SPLINE
SPL {X   -94.059, Y  +248.080, Z    +0.000, E1   +58.275, E3 +53997.383}
SPL {X  -130.769, Y  +285.325, Z    +0.000, E1   +56.495, E3 +54037.260}
SPL {X  -149.689, Y  +321.019, Z    +0.000, E1   +46.817, E3 +54049.344}
SPL {X  -157.484, Y  +349.293, Z    +0.000, E1   +30.654, E3 +54053.637}
SPL {X  -159.556, Y  +365.719, Z    +0.000, E1   +15.845, E3 +54054.829}
SPL {X  -159.982, Y  +375.924, Z    +0.000, E1    +4.476, E3 +54055.131}
SPL {X  -159.990, Y  +379.531, Z    +0.000, E1    -0.039, E3 +54055.158}
SPL {X  -159.990, Y  +382.420, Z    +0.000, E1    -7.600, E3 +54055.186}
SPL {X  -159.990, Y  +386.504, Z    +0.000, E1   -19.860, E3 +54055.292}
SPL {X  -159.990, Y  +392.530, Z    +0.000, E1   -36.133, E3 +54055.607}
SPL {X  -159.990, Y  +400.492, Z    +0.000, E1   -51.837, E3 +54056.260}
SPL {X  -159.990, Y  +409.662, Z    +0.000, E1   -61.705, E3 +54057.371}
SPL {X  -159.990, Y  +434.697, Z    +0.000, E1   -71.504, E3 +54062.391}
SPL {X  -159.990, Y  +521.523, Z    +0.000, E1   -76.035, E3 +54088.671}
SPL {X  -154.459, Y  +718.205, Z    +0.000, E1   -76.329, E3 +54170.467}
SPL {X  -151.356, Y  +728.349, Z    +0.000, E1   -76.056, E3 +54178.682}
SPL {X  -147.124, Y  +739.360, Z    +0.000, E1   -75.690, E3 +54188.278}
SPL {X  -142.861, Y  +748.524, Z    +0.000, E1   -75.261, E3 +54196.963}
SPL {X  -138.117, Y  +757.250, Z    +0.000, E1   -74.803, E3 +54205.567}
SPL {X  -133.491, Y  +764.686, Z    +0.000, E1   -74.276, E3 +54213.308}
SPL {X  -128.839, Y  +771.354, Z    +0.000, E1   -73.759, E3 +54220.326}
SPL {X  -124.765, Y  +776.652, Z    +0.000, E1   -73.233, E3 +54225.976}
SPL {X  -121.376, Y  +780.734, Z    +0.000, E1   -72.804, E3 +54230.238}
SPL {X  -118.281, Y  +784.233, Z    +0.000, E1   -72.371, E3 +54233.806}
SPL {X   -72.391, Y  +819.176, Z    +0.000, E1   -59.867, E3 +54329.692}
ENDSPLINE

SPLINE
SPL {X  -116.241, Y  +786.431, Z    +0.000, E1   -57.120, E3 +54554.134}
SPL {X  -148.710, Y  +735.509, Z    +0.000, E1   -46.282, E3 +54579.867}
SPL {X  -157.559, Y  +704.285, Z    +0.000, E1   -29.037, E3 +54585.196}
SPL {X  -159.709, Y  +685.986, Z    +0.000, E1   -12.810, E3 +54586.528}
SPL {X  -159.990, Y  +674.648, Z    +0.000, E1    -0.349, E3 +54586.787}
SPL {X  -159.990, Y  +672.787, Z    +0.000, E1    +4.022, E3 +54586.800}
SPL {X  -159.990, Y  +669.267, Z    +0.000, E1   +13.665, E3 +54586.870}
SPL {X  -159.990, Y  +663.438, Z    +0.000, E1   +29.379, E3 +54587.141}
SPL {X  -159.990, Y  +655.264, Z    +0.000, E1   +47.291, E3 +54587.758}
SPL {X  -159.990, Y  +645.368, Z    +0.000, E1   +59.257, E3 +54589.001}
SPL {X  -159.990, Y  +624.023, Z    +0.000, E1   +69.513, E3 +54593.126}
SPL {X  -159.990, Y  +543.075, Z    +0.000, E1   +75.590, E3 +54616.774}
SPL {X  -156.121, Y  +342.530, Z    +0.000, E1   +75.868, E3 +54703.420}
SPL {X  -153.498, Y  +332.386, Z    +0.000, E1   +75.628, E3 +54711.425}
ENDSPLINE

SPLINE
SPL {X  -155.252, Y  +338.851, Z    +0.000, E1   +74.632, E3 +54718.803}
SPL {X  -159.103, Y  +360.678, Z    +0.000, E1   +72.233, E3 +54731.128}
ENDSPLINE

SPLINE
SPL {X  -154.371, Y  +335.471, Z    +0.000, E1   +73.016, E3 +54739.698}
SPL {X  -149.938, Y  +321.685, Z    +0.000, E1   +73.398, E3 +54744.393}
SPL {X  -145.016, Y  +309.920, Z    +0.000, E1   +73.647, E3 +54748.914}
SPL {X  -136.944, Y  +294.777, Z    +0.000, E1   +74.219, E3 +54752.215}
SPL {X  -132.590, Y  +287.964, Z    +0.000, E1   +73.910, E3 +54757.960}
SPL {X  -129.541, Y  +283.606, Z    +0.000, E1   +73.551, E3 +54762.600}
SPL {X  -125.403, Y  +278.147, Z    +0.000, E1   +73.063, E3 +54768.407}
SPL {X  -121.908, Y  +273.889, Z    +0.000, E1   +72.578, E3 +54772.954}
SPL {X  -119.156, Y  +270.736, Z    +0.000, E1   +72.213, E3 +54776.204}
SPL {X  -117.531, Y  +268.949, Z    +0.000, E1   +71.964, E3 +54778.019}
SPL {X   -74.907, Y  +236.129, Z    +0.000, E1   +61.720, E3 +54855.055}
ENDSPLINE

SPLINE
SPL {X   -94.059, Y  +248.080, Z    +0.000, E1   +58.275, E3 +55076.748}
SPL {X  -130.769, Y  +285.325, Z    +0.000, E1   +56.495, E3 +55116.625}
SPL {X  -149.689, Y  +321.019, Z    +0.000, E1   +46.817, E3 +55128.709}
SPL {X  -155.950, Y  +341.772, Z    +0.000, E1   +35.915, E3 +55132.208}
SPL {X  -158.168, Y  +353.421, Z    +0.000, E1   +27.296, E3 +55133.393}
SPL {X  -159.556, Y  +365.719, Z    +0.000, E1   +15.845, E3 +55134.194}
SPL {X  -159.982, Y  +375.924, Z    +0.000, E1    +4.476, E3 +55134.496}
SPL {X  -159.990, Y  +379.800, Z    +0.000, E1    -0.377, E3 +55134.524}
SPL {X  -159.990, Y  +383.422, Z    +0.000, E1   -10.730, E3 +55134.567}
SPL {X  -159.990, Y  +387.978, Z    +0.000, E1   -23.882, E3 +55134.720}
SPL {X  -159.990, Y  +394.494, Z    +0.000, E1   -40.961, E3 +55135.101}
SPL {X  -159.990, Y  +400.492, Z    +0.000, E1   -51.837, E3 +55135.625}
SPL {X  -159.990, Y  +409.662, Z    +0.000, E1   -61.705, E3 +55136.736}
SPL {X  -159.990, Y  +434.697, Z    +0.000, E1   -71.504, E3 +55141.756}
SPL {X  -159.990, Y  +521.523, Z    +0.000, E1   -76.035, E3 +55168.036}
SPL {X  -154.459, Y  +718.205, Z    +0.000, E1   -76.329, E3 +55249.832}
SPL {X  -151.356, Y  +728.349, Z    +0.000, E1   -76.056, E3 +55258.047}
SPL {X  -147.124, Y  +739.360, Z    +0.000, E1   -75.690, E3 +55267.644}
SPL {X  -142.861, Y  +748.524, Z    +0.000, E1   -75.261, E3 +55276.328}
SPL {X  -138.117, Y  +757.250, Z    +0.000, E1   -74.803, E3 +55284.932}
SPL {X  -133.491, Y  +764.686, Z    +0.000, E1   -74.276, E3 +55292.673}
SPL {X  -130.530, Y  +769.013, Z    +0.000, E1   -73.929, E3 +55297.255}
SPL {X  -127.734, Y  +772.837, Z    +0.000, E1   -73.601, E3 +55301.307}
SPL {X  -124.765, Y  +776.652, Z    +0.000, E1   -73.233, E3 +55305.341}
SPL {X  -121.376, Y  +780.734, Z    +0.000, E1   -72.804, E3 +55309.603}
SPL {X  -118.281, Y  +784.233, Z    +0.000, E1   -72.371, E3 +55313.171}
SPL {X   -72.391, Y  +819.176, Z    +0.000, E1   -59.867, E3 +55409.057}
ENDSPLINE

SPLINE
SPL {X  -116.241, Y  +786.431, Z    +0.000, E1   -57.120, E3 +55633.499}
SPL {X  -148.710, Y  +735.509, Z    +0.000, E1   -46.282, E3 +55659.232}
SPL {X  -157.559, Y  +704.285, Z    +0.000, E1   -29.037, E3 +55664.561}
SPL {X  -159.430, Y  +689.871, Z    +0.000, E1   -16.582, E3 +55665.711}
SPL {X  -159.960, Y  +679.609, Z    +0.000, E1    -6.021, E3 +55666.094}
SPL {X  -159.990, Y  +674.508, Z    +0.000, E1    -0.018, E3 +55666.153}
SPL {X  -159.990, Y  +672.787, Z    +0.000, E1    +4.022, E3 +55666.165}
SPL {X  -159.990, Y  +669.267, Z    +0.000, E1   +13.665, E3 +55666.235}
SPL {X  -159.990, Y  +663.438, Z    +0.000, E1   +29.379, E3 +55666.506}
SPL {X  -159.990, Y  +655.264, Z    +0.000, E1   +47.291, E3 +55667.123}
SPL {X  -159.990, Y  +645.368, Z    +0.000, E1   +59.257, E3 +55668.366}
SPL {X  -159.990, Y  +624.023, Z    +0.000, E1   +69.513, E3 +55672.491}
SPL {X  -159.990, Y  +543.075, Z    +0.000, E1   +75.590, E3 +55696.139}
SPL {X  -156.121, Y  +342.530, Z    +0.000, E1   +75.868, E3 +55782.785}
SPL {X  -153.498, Y  +332.386, Z    +0.000, E1   +75.628, E3 +55790.790}
ENDSPLINE

SPLINE
SPL {X  -155.252, Y  +338.851, Z    +0.000, E1   +74.632, E3 +55798.168}
SPL {X  -159.103, Y  +360.678, Z    +0.000, E1   +72.233, E3 +55810.493}
ENDSPLINE

SPLINE
SPL {X  -154.371, Y  +335.471, Z    +0.000, E1   +73.016, E3 +55819.064}
SPL {X  -149.938, Y  +321.685, Z    +0.000, E1   +73.398, E3 +55823.758}
SPL {X  -145.016, Y  +309.920, Z    +0.000, E1   +73.647, E3 +55828.279}
SPL {X  -139.138, Y  +298.522, Z    +0.000, E1   +74.138, E3 +55830.295}
SPL {X  -135.697, Y  +292.747, Z    +0.000, E1   +74.259, E3 +55832.297}
SPL {X  -132.590, Y  +287.964, Z    +0.000, E1   +73.910, E3 +55837.325}
SPL {X  -129.541, Y  +283.606, Z    +0.000, E1   +73.551, E3 +55841.965}
SPL {X  -126.457, Y  +279.493, Z    +0.000, E1   +73.175, E3 +55846.364}
SPL {X  -122.770, Y  +274.912, Z    +0.000, E1   +72.712, E3 +55851.220}
SPL {X  -119.156, Y  +270.736, Z    +0.000, E1   +72.213, E3 +55855.569}
SPL {X  -117.531, Y  +268.949, Z    +0.000, E1   +71.964, E3 +55857.384}
SPL {X   -74.907, Y  +236.129, Z    +0.000, E1   +61.720, E3 +55934.420}
ENDSPLINE

SPLINE
SPL {X   -94.059, Y  +248.080, Z    +0.000, E1   +58.275, E3 +56156.113}
SPL {X  -130.769, Y  +285.325, Z    +0.000, E1   +56.495, E3 +56195.990}
SPL {X  -149.689, Y  +321.019, Z    +0.000, E1   +46.817, E3 +56208.074}
SPL {X  -157.484, Y  +349.293, Z    +0.000, E1   +30.654, E3 +56212.367}
SPL {X  -159.556, Y  +365.719, Z    +0.000, E1   +15.845, E3 +56213.559}
SPL {X  -159.982, Y  +375.924, Z    +0.000, E1    +4.476, E3 +56213.861}
SPL {X  -159.990, Y  +379.531, Z    +0.000, E1    -0.039, E3 +56213.888}
SPL {X  -159.990, Y  +382.420, Z    +0.000, E1    -7.600, E3 +56213.916}
SPL {X  -159.990, Y  +386.504, Z    +0.000, E1   -19.860, E3 +56214.022}
SPL {X  -159.990, Y  +392.530, Z    +0.000, E1   -36.133, E3 +56214.337}
SPL {X  -159.990, Y  +400.492, Z    +0.000, E1   -51.837, E3 +56214.990}
SPL {X  -159.990, Y  +409.662, Z    +0.000, E1   -61.705, E3 +56216.101}
SPL {X  -159.990, Y  +434.697, Z    +0.000, E1   -71.504, E3 +56221.121}
SPL {X  -159.990, Y  +521.523, Z    +0.000, E1   -76.035, E3 +56247.401}
SPL {X  -154.459, Y  +718.205, Z    +0.000, E1   -76.329, E3 +56329.197}
SPL {X  -151.356, Y  +728.349, Z    +0.000, E1   -76.056, E3 +56337.412}
SPL {X  -148.399, Y  +736.287, Z    +0.000, E1   -75.788, E3 +56344.291}
SPL {X  -144.005, Y  +746.209, Z    +0.000, E1   -75.396, E3 +56353.407}
SPL {X  -138.117, Y  +757.250, Z    +0.000, E1   -74.803, E3 +56364.297}
SPL {X  -133.491, Y  +764.686, Z    +0.000, E1   -74.276, E3 +56372.038}
SPL {X  -128.839, Y  +771.354, Z    +0.000, E1   -73.759, E3 +56379.057}
SPL {X  -123.568, Y  +778.125, Z    +0.000, E1   -73.105, E3 +56386.228}
SPL {X  -118.985, Y  +783.455, Z    +0.000, E1   -72.490, E3 +56391.736}
SPL {X   -72.391, Y  +819.176, Z    +0.000, E1   -59.867, E3 +56488.422}
ENDSPLINE

SPLINE
SPL {X   -92.809, Y  +806.820, Z    +0.000, E1   -56.994, E3 +56681.217}
SPL {X  -120.521, Y  +781.721, Z    +0.000, E1   -56.766, E3 +56717.316}
SPL {X  -143.482, Y  +747.279, Z    +0.000, E1   -50.227, E3 +56735.329}
SPL {X  -154.118, Y  +719.449, Z    +0.000, E1   -38.836, E3 +56741.908}
SPL {X  -158.958, Y  +694.646, Z    +0.000, E1   -21.132, E3 +56744.760}
SPL {X  -159.960, Y  +679.609, Z    +0.000, E1    -6.021, E3 +56745.460}
SPL {X  -159.990, Y  +674.508, Z    +0.000, E1    -0.018, E3 +56745.518}
SPL {X  -159.990, Y  +672.787, Z    +0.000, E1    +4.022, E3 +56745.530}
SPL {X  -159.990, Y  +669.267, Z    +0.000, E1   +13.665, E3 +56745.600}
SPL {X  -159.990, Y  +663.438, Z    +0.000, E1   +29.379, E3 +56745.871}
SPL {X  -159.990, Y  +655.264, Z    +0.000, E1   +47.291, E3 +56746.488}
SPL {X  -159.990, Y  +645.368, Z    +0.000, E1   +59.257, E3 +56747.731}
SPL {X  -159.990, Y  +624.023, Z    +0.000, E1   +69.513, E3 +56751.856}
SPL {X  -159.990, Y  +543.075, Z    +0.000, E1   +75.590, E3 +56775.504}
SPL {X  -156.121, Y  +342.530, Z    +0.000, E1   +75.868, E3 +56862.150}
SPL {X  -153.498, Y  +332.386, Z    +0.000, E1   +75.628, E3 +56870.155}
ENDSPLINE

SPLINE
SPL {X  -155.252, Y  +338.851, Z    +0.000, E1   +74.632, E3 +56877.533}
SPL {X  -159.103, Y  +360.678, Z    +0.000, E1   +72.233, E3 +56889.858}
ENDSPLINE

SPLINE
SPL {X  -154.371, Y  +335.471, Z    +0.000, E1   +73.016, E3 +56898.429}
SPL {X  -149.938, Y  +321.685, Z    +0.000, E1   +73.398, E3 +56903.123}
SPL {X  -145.016, Y  +309.920, Z    +0.000, E1   +73.647, E3 +56907.644}
SPL {X  -139.138, Y  +298.522, Z    +0.000, E1   +74.138, E3 +56909.660}
SPL {X  -135.697, Y  +292.747, Z    +0.000, E1   +74.259, E3 +56911.662}
SPL {X  -132.590, Y  +287.964, Z    +0.000, E1   +73.910, E3 +56916.690}
SPL {X  -129.541, Y  +283.606, Z    +0.000, E1   +73.551, E3 +56921.330}
SPL {X  -126.457, Y  +279.493, Z    +0.000, E1   +73.175, E3 +56925.729}
SPL {X  -122.770, Y  +274.912, Z    +0.000, E1   +72.712, E3 +56930.585}
SPL {X  -118.941, Y  +270.496, Z    +0.000, E1   +72.188, E3 +56935.172}
SPL {X   -74.907, Y  +236.129, Z    +0.000, E1   +61.720, E3 +57013.785}
ENDSPLINE

SPLINE
SPL {X   -94.059, Y  +248.080, Z    +0.000, E1   +58.275, E3 +57235.478}
SPL {X  -136.558, Y  +294.141, Z    +0.000, E1   +54.887, E3 +57279.333}
SPL {X  -151.843, Y  +327.098, Z    +0.000, E1   +44.118, E3 +57288.692}
SPL {X  -157.484, Y  +349.293, Z    +0.000, E1   +30.654, E3 +57291.732}
SPL {X  -159.556, Y  +365.719, Z    +0.000, E1   +15.845, E3 +57292.924}
SPL {X  -159.982, Y  +375.924, Z    +0.000, E1    +4.476, E3 +57293.226}
SPL {X  -159.990, Y  +379.531, Z    +0.000, E1    -0.039, E3 +57293.253}
SPL {X  -159.990, Y  +382.420, Z    +0.000, E1    -7.600, E3 +57293.281}
SPL {X  -159.990, Y  +386.504, Z    +0.000, E1   -19.860, E3 +57293.387}
SPL {X  -159.990, Y  +392.530, Z    +0.000, E1   -36.133, E3 +57293.702}
SPL {X  -159.990, Y  +400.492, Z    +0.000, E1   -51.837, E3 +57294.355}
SPL {X  -159.990, Y  +409.662, Z    +0.000, E1   -61.705, E3 +57295.466}
SPL {X  -159.990, Y  +434.697, Z    +0.000, E1   -71.504, E3 +57300.486}
SPL {X  -159.990, Y  +521.523, Z    +0.000, E1   -76.035, E3 +57326.767}
SPL {X  -154.459, Y  +718.205, Z    +0.000, E1   -76.329, E3 +57408.562}
SPL {X  -151.356, Y  +728.349, Z    +0.000, E1   -76.056, E3 +57416.777}
SPL {X  -148.399, Y  +736.287, Z    +0.000, E1   -75.788, E3 +57423.656}
SPL {X  -144.005, Y  +746.209, Z    +0.000, E1   -75.396, E3 +57432.772}
SPL {X  -138.117, Y  +757.250, Z    +0.000, E1   -74.803, E3 +57443.662}
SPL {X  -133.491, Y  +764.686, Z    +0.000, E1   -74.276, E3 +57451.403}
SPL {X  -128.839, Y  +771.354, Z    +0.000, E1   -73.759, E3 +57458.422}
SPL {X  -123.568, Y  +778.125, Z    +0.000, E1   -73.105, E3 +57465.593}
SPL {X  -118.985, Y  +783.455, Z    +0.000, E1   -72.490, E3 +57471.101}
SPL {X   -72.391, Y  +819.176, Z    +0.000, E1   -59.867, E3 +57567.787}
ENDSPLINE

SPLINE
SPL {X   -92.809, Y  +806.820, Z    +0.000, E1   -56.994, E3 +57760.582}
SPL {X  -120.521, Y  +781.721, Z    +0.000, E1   -56.766, E3 +57796.681}
SPL {X  -148.710, Y  +735.509, Z    +0.000, E1   -46.282, E3 +57817.962}
SPL {X  -157.559, Y  +704.285, Z    +0.000, E1   -29.037, E3 +57823.291}
SPL {X  -159.430, Y  +689.871, Z    +0.000, E1   -16.582, E3 +57824.442}
SPL {X  -159.960, Y  +679.609, Z    +0.000, E1    -6.021, E3 +57824.825}
SPL {X  -159.990, Y  +674.508, Z    +0.000, E1    -0.018, E3 +57824.883}
SPL {X  -159.990, Y  +672.787, Z    +0.000, E1    +4.022, E3 +57824.895}
SPL {X  -159.990, Y  +669.267, Z    +0.000, E1   +13.665, E3 +57824.965}
SPL {X  -159.990, Y  +663.438, Z    +0.000, E1   +29.379, E3 +57825.236}
SPL {X  -159.990, Y  +655.264, Z    +0.000, E1   +47.291, E3 +57825.853}
SPL {X  -159.990, Y  +645.368, Z    +0.000, E1   +59.257, E3 +57827.096}
SPL {X  -159.990, Y  +624.023, Z    +0.000, E1   +69.513, E3 +57831.221}
SPL {X  -159.990, Y  +543.075, Z    +0.000, E1   +75.590, E3 +57854.869}
SPL {X  -156.121, Y  +342.530, Z    +0.000, E1   +75.868, E3 +57941.515}
SPL {X  -153.865, Y  +333.657, Z    +0.000, E1   +75.438, E3 +57951.119}
ENDSPLINE

SPLINE
SPL {X  -159.644, Y  +366.989, Z    +0.000, E1   +72.058, E3 +57966.646}
ENDSPLINE

SPLINE
SPL {X  -156.933, Y  +346.374, Z    +0.000, E1   +72.645, E3 +57974.535}
SPL {X  -151.144, Y  +325.039, Z    +0.000, E1   +73.323, E3 +57981.215}
SPL {X  -145.016, Y  +309.920, Z    +0.000, E1   +73.647, E3 +57987.009}
SPL {X  -136.944, Y  +294.777, Z    +0.000, E1   +74.219, E3 +57990.311}
SPL {X  -132.590, Y  +287.964, Z    +0.000, E1   +73.910, E3 +57996.055}
SPL {X  -129.541, Y  +283.606, Z    +0.000, E1   +73.551, E3 +58000.695}
SPL {X  -125.403, Y  +278.147, Z    +0.000, E1   +73.063, E3 +58006.503}
SPL {X  -121.908, Y  +273.889, Z    +0.000, E1   +72.578, E3 +58011.049}
SPL {X  -118.941, Y  +270.496, Z    +0.000, E1   +72.188, E3 +58014.537}
SPL {X   -74.907, Y  +236.129, Z    +0.000, E1   +61.720, E3 +58093.150}
ENDSPLINE

SPLINE
SPL {X   -94.059, Y  +248.080, Z    +0.000, E1   +58.275, E3 +58314.843}
SPL {X  -136.558, Y  +294.141, Z    +0.000, E1   +54.887, E3 +58358.698}
SPL {X  -151.843, Y  +327.098, Z    +0.000, E1   +44.118, E3 +58368.058}
SPL {X  -157.484, Y  +349.293, Z    +0.000, E1   +30.654, E3 +58371.097}
SPL {X  -159.556, Y  +365.719, Z    +0.000, E1   +15.845, E3 +58372.289}
SPL {X  -159.982, Y  +375.924, Z    +0.000, E1    +4.476, E3 +58372.591}
SPL {X  -159.990, Y  +379.531, Z    +0.000, E1    -0.039, E3 +58372.618}
SPL {X  -159.990, Y  +382.420, Z    +0.000, E1    -7.600, E3 +58372.647}
SPL {X  -159.990, Y  +386.504, Z    +0.000, E1   -19.860, E3 +58372.752}
SPL {X  -159.990, Y  +392.530, Z    +0.000, E1   -36.133, E3 +58373.067}
SPL {X  -159.990, Y  +400.492, Z    +0.000, E1   -51.837, E3 +58373.720}
SPL {X  -159.990, Y  +409.662, Z    +0.000, E1   -61.705, E3 +58374.831}
SPL {X  -159.990, Y  +434.697, Z    +0.000, E1   -71.504, E3 +58379.851}
SPL {X  -159.990, Y  +521.523, Z    +0.000, E1   -76.035, E3 +58406.132}
SPL {X  -154.459, Y  +718.205, Z    +0.000, E1   -76.329, E3 +58487.927}
SPL {X  -151.356, Y  +728.349, Z    +0.000, E1   -76.056, E3 +58496.143}
SPL {X  -148.399, Y  +736.287, Z    +0.000, E1   -75.788, E3 +58503.021}
SPL {X  -144.005, Y  +746.209, Z    +0.000, E1   -75.396, E3 +58512.137}
SPL {X  -138.117, Y  +757.250, Z    +0.000, E1   -74.803, E3 +58523.027}
SPL {X  -133.491, Y  +764.686, Z    +0.000, E1   -74.276, E3 +58530.768}
SPL {X  -128.839, Y  +771.354, Z    +0.000, E1   -73.759, E3 +58537.787}
SPL {X  -123.568, Y  +778.125, Z    +0.000, E1   -73.105, E3 +58544.958}
SPL {X  -118.985, Y  +783.455, Z    +0.000, E1   -72.490, E3 +58550.466}
SPL {X   -72.391, Y  +819.176, Z    +0.000, E1   -59.867, E3 +58647.152}
ENDSPLINE

SPLINE
SPL {X   -92.809, Y  +806.820, Z    +0.000, E1   -56.994, E3 +58839.947}
SPL {X  -120.521, Y  +781.721, Z    +0.000, E1   -56.766, E3 +58876.046}
SPL {X  -143.482, Y  +747.279, Z    +0.000, E1   -50.227, E3 +58894.059}
SPL {X  -154.118, Y  +719.449, Z    +0.000, E1   -38.836, E3 +58900.638}
SPL {X  -158.958, Y  +694.646, Z    +0.000, E1   -21.132, E3 +58903.490}
SPL {X  -159.960, Y  +679.609, Z    +0.000, E1    -6.021, E3 +58904.190}
SPL {X  -159.990, Y  +674.508, Z    +0.000, E1    -0.018, E3 +58904.248}
SPL {X  -159.990, Y  +672.787, Z    +0.000, E1    +4.022, E3 +58904.260}
SPL {X  -159.990, Y  +669.267, Z    +0.000, E1   +13.665, E3 +58904.330}
SPL {X  -159.990, Y  +663.438, Z    +0.000, E1   +29.379, E3 +58904.601}
SPL {X  -159.990, Y  +655.264, Z    +0.000, E1   +47.291, E3 +58905.218}
SPL {X  -159.990, Y  +645.368, Z    +0.000, E1   +59.257, E3 +58906.461}
SPL {X  -159.990, Y  +624.023, Z    +0.000, E1   +69.513, E3 +58910.586}
SPL {X  -159.990, Y  +543.075, Z    +0.000, E1   +75.590, E3 +58934.234}
SPL {X  -156.121, Y  +342.530, Z    +0.000, E1   +75.868, E3 +59020.880}
SPL {X  -153.498, Y  +332.386, Z    +0.000, E1   +75.628, E3 +59028.885}
ENDSPLINE

SPLINE
SPL {X  -155.252, Y  +338.851, Z    +0.000, E1   +74.632, E3 +59036.263}
SPL {X  -159.103, Y  +360.678, Z    +0.000, E1   +72.233, E3 +59048.588}
ENDSPLINE

SPLINE
SPL {X  -154.371, Y  +335.471, Z    +0.000, E1   +73.016, E3 +59057.159}
SPL {X  -149.938, Y  +321.685, Z    +0.000, E1   +73.398, E3 +59061.853}
SPL {X  -145.016, Y  +309.920, Z    +0.000, E1   +73.647, E3 +59066.374}
SPL {X  -139.138, Y  +298.522, Z    +0.000, E1   +74.138, E3 +59068.390}
SPL {X  -135.697, Y  +292.747, Z    +0.000, E1   +74.259, E3 +59070.392}
SPL {X  -132.590, Y  +287.964, Z    +0.000, E1   +73.910, E3 +59075.420}
SPL {X  -129.541, Y  +283.606, Z    +0.000, E1   +73.551, E3 +59080.061}
SPL {X  -126.457, Y  +279.493, Z    +0.000, E1   +73.175, E3 +59084.460}
SPL {X  -122.770, Y  +274.912, Z    +0.000, E1   +72.712, E3 +59089.315}
SPL {X  -118.941, Y  +270.496, Z    +0.000, E1   +72.188, E3 +59093.902}
SPL {X   -74.907, Y  +236.129, Z    +0.000, E1   +61.720, E3 +59172.516}
ENDSPLINE

SPLINE
SPL {X   -94.059, Y  +248.080, Z    +0.000, E1   +58.275, E3 +59394.209}
SPL {X  -136.558, Y  +294.141, Z    +0.000, E1   +54.887, E3 +59438.063}
SPL {X  -151.843, Y  +327.098, Z    +0.000, E1   +44.118, E3 +59447.423}
SPL {X  -157.484, Y  +349.293, Z    +0.000, E1   +30.654, E3 +59450.462}
SPL {X  -159.556, Y  +365.719, Z    +0.000, E1   +15.845, E3 +59451.655}
SPL {X  -159.982, Y  +375.924, Z    +0.000, E1    +4.476, E3 +59451.956}
SPL {X  -159.990, Y  +379.531, Z    +0.000, E1    -0.039, E3 +59451.983}
SPL {X  -159.990, Y  +382.420, Z    +0.000, E1    -7.600, E3 +59452.012}
SPL {X  -159.990, Y  +386.504, Z    +0.000, E1   -19.860, E3 +59452.117}
SPL {X  -159.990, Y  +392.530, Z    +0.000, E1   -36.133, E3 +59452.432}
SPL {X  -159.990, Y  +400.492, Z    +0.000, E1   -51.837, E3 +59453.085}
SPL {X  -159.990, Y  +409.662, Z    +0.000, E1   -61.705, E3 +59454.196}
SPL {X  -159.990, Y  +434.697, Z    +0.000, E1   -71.504, E3 +59459.216}
SPL {X  -159.990, Y  +521.523, Z    +0.000, E1   -76.035, E3 +59485.497}
SPL {X  -154.459, Y  +718.205, Z    +0.000, E1   -76.329, E3 +59567.292}
SPL {X  -151.356, Y  +728.349, Z    +0.000, E1   -76.056, E3 +59575.508}
SPL {X  -148.399, Y  +736.287, Z    +0.000, E1   -75.788, E3 +59582.386}
SPL {X  -144.005, Y  +746.209, Z    +0.000, E1   -75.396, E3 +59591.502}
SPL {X  -138.117, Y  +757.250, Z    +0.000, E1   -74.803, E3 +59602.392}
SPL {X  -133.491, Y  +764.686, Z    +0.000, E1   -74.276, E3 +59610.133}
SPL {X  -128.839, Y  +771.354, Z    +0.000, E1   -73.759, E3 +59617.152}
SPL {X  -123.568, Y  +778.125, Z    +0.000, E1   -73.105, E3 +59624.324}
SPL {X  -118.985, Y  +783.455, Z    +0.000, E1   -72.490, E3 +59629.831}
SPL {X   -72.391, Y  +819.176, Z    +0.000, E1   -59.867, E3 +59726.517}
ENDSPLINE

SPLINE
SPL {X   -92.809, Y  +806.820, Z    +0.000, E1   -56.994, E3 +59919.312}
SPL {X  -120.521, Y  +781.721, Z    +0.000, E1   -56.766, E3 +59955.411}
SPL {X  -148.710, Y  +735.509, Z    +0.000, E1   -46.282, E3 +59976.692}
SPL {X  -157.559, Y  +704.285, Z    +0.000, E1   -29.037, E3 +59982.022}
SPL {X  -159.430, Y  +689.871, Z    +0.000, E1   -16.582, E3 +59983.172}
SPL {X  -159.960, Y  +679.609, Z    +0.000, E1    -6.021, E3 +59983.555}
SPL {X  -159.990, Y  +674.508, Z    +0.000, E1    -0.018, E3 +59983.613}
SPL {X  -159.990, Y  +672.787, Z    +0.000, E1    +4.022, E3 +59983.625}
SPL {X  -159.990, Y  +669.267, Z    +0.000, E1   +13.665, E3 +59983.695}
SPL {X  -159.990, Y  +663.438, Z    +0.000, E1   +29.379, E3 +59983.966}
SPL {X  -159.990, Y  +655.264, Z    +0.000, E1   +47.291, E3 +59984.583}
SPL {X  -159.990, Y  +645.368, Z    +0.000, E1   +59.257, E3 +59985.826}
SPL {X  -159.990, Y  +624.023, Z    +0.000, E1   +69.513, E3 +59989.951}
SPL {X  -159.990, Y  +543.075, Z    +0.000, E1   +75.590, E3 +60013.599}
SPL {X  -156.121, Y  +342.530, Z    +0.000, E1   +75.868, E3 +60100.245}
SPL {X  -153.865, Y  +333.657, Z    +0.000, E1   +75.438, E3 +60109.849}
ENDSPLINE

SPLINE
SPL {X  -159.644, Y  +366.989, Z    +0.000, E1   +72.058, E3 +60125.376}
ENDSPLINE

SPLINE
SPL {X  -156.933, Y  +346.374, Z    +0.000, E1   +72.645, E3 +60133.266}
SPL {X  -151.144, Y  +325.039, Z    +0.000, E1   +73.323, E3 +60139.945}
SPL {X  -146.668, Y  +313.584, Z    +0.000, E1   +73.560, E3 +60144.427}
SPL {X  -141.230, Y  +302.327, Z    +0.000, E1   +73.933, E3 +60147.399}
SPL {X  -135.697, Y  +292.747, Z    +0.000, E1   +74.259, E3 +60149.757}
SPL {X  -132.590, Y  +287.964, Z    +0.000, E1   +73.910, E3 +60154.785}
SPL {X  -129.541, Y  +283.606, Z    +0.000, E1   +73.551, E3 +60159.426}
SPL {X  -125.403, Y  +278.147, Z    +0.000, E1   +73.063, E3 +60165.233}
SPL {X  -121.908, Y  +273.889, Z    +0.000, E1   +72.578, E3 +60169.779}
SPL {X  -119.156, Y  +270.736, Z    +0.000, E1   +72.213, E3 +60173.029}
SPL {X  -117.531, Y  +268.949, Z    +0.000, E1   +71.964, E3 +60174.845}
SPL {X   -74.907, Y  +236.129, Z    +0.000, E1   +61.720, E3 +60251.881}
ENDSPLINE

SPLINE
SPL {X   -94.059, Y  +248.080, Z    +0.000, E1   +58.275, E3 +60473.574}
SPL {X  -130.769, Y  +285.325, Z    +0.000, E1   +56.495, E3 +60513.451}
SPL {X  -149.689, Y  +321.019, Z    +0.000, E1   +46.817, E3 +60525.535}
SPL {X  -157.484, Y  +349.293, Z    +0.000, E1   +30.654, E3 +60529.827}
SPL {X  -159.556, Y  +365.719, Z    +0.000, E1   +15.845, E3 +60531.020}
SPL {X  -159.982, Y  +375.924, Z    +0.000, E1    +4.476, E3 +60531.321}
SPL {X  -159.990, Y  +379.531, Z    +0.000, E1    -0.039, E3 +60531.348}
SPL {X  -159.990, Y  +382.420, Z    +0.000, E1    -7.600, E3 +60531.377}
SPL {X  -159.990, Y  +386.504, Z    +0.000, E1   -19.860, E3 +60531.482}
SPL {X  -159.990, Y  +392.530, Z    +0.000, E1   -36.133, E3 +60531.797}
SPL {X  -159.990, Y  +400.492, Z    +0.000, E1   -51.837, E3 +60532.450}
SPL {X  -159.990, Y  +409.662, Z    +0.000, E1   -61.705, E3 +60533.561}
SPL {X  -159.990, Y  +434.697, Z    +0.000, E1   -71.504, E3 +60538.581}
SPL {X  -159.990, Y  +521.523, Z    +0.000, E1   -76.035, E3 +60564.862}
SPL {X  -154.459, Y  +718.205, Z    +0.000, E1   -76.329, E3 +60646.657}
SPL {X  -151.356, Y  +728.349, Z    +0.000, E1   -76.056, E3 +60654.873}
SPL {X  -147.124, Y  +739.360, Z    +0.000, E1   -75.690, E3 +60664.469}
SPL {X  -142.861, Y  +748.524, Z    +0.000, E1   -75.261, E3 +60673.154}
SPL {X  -139.796, Y  +754.307, Z    +0.000, E1   -74.951, E3 +60678.842}
SPL {X  -136.850, Y  +759.378, Z    +0.000, E1   -74.643, E3 +60683.986}
SPL {X  -133.491, Y  +764.686, Z    +0.000, E1   -74.276, E3 +60689.498}
SPL {X  -130.530, Y  +769.013, Z    +0.000, E1   -73.929, E3 +60694.080}
SPL {X  -127.734, Y  +772.837, Z    +0.000, E1   -73.601, E3 +60698.132}
SPL {X  -124.765, Y  +776.652, Z    +0.000, E1   -73.233, E3 +60702.167}
SPL {X  -121.376, Y  +780.734, Z    +0.000, E1   -72.804, E3 +60706.428}
SPL {X  -118.281, Y  +784.233, Z    +0.000, E1   -72.371, E3 +60709.997}
SPL {X   -72.391, Y  +819.176, Z    +0.000, E1   -59.867, E3 +60805.882}
ENDSPLINE

SPLINE
SPL {X  -116.241, Y  +786.431, Z    +0.000, E1   -57.120, E3 +61030.325}
SPL {X  -143.482, Y  +747.279, Z    +0.000, E1   -50.227, E3 +61052.789}
SPL {X  -154.118, Y  +719.449, Z    +0.000, E1   -38.836, E3 +61059.369}
SPL {X  -158.958, Y  +694.646, Z    +0.000, E1   -21.132, E3 +61062.220}
SPL {X  -159.960, Y  +679.609, Z    +0.000, E1    -6.021, E3 +61062.920}
SPL {X  -159.990, Y  +674.508, Z    +0.000, E1    -0.018, E3 +61062.979}
SPL {X  -159.990, Y  +672.787, Z    +0.000, E1    +4.022, E3 +61062.990}
SPL {X  -159.990, Y  +669.267, Z    +0.000, E1   +13.665, E3 +61063.061}
SPL {X  -159.990, Y  +663.438, Z    +0.000, E1   +29.379, E3 +61063.331}
SPL {X  -159.990, Y  +655.264, Z    +0.000, E1   +47.291, E3 +61063.948}
SPL {X  -159.990, Y  +645.368, Z    +0.000, E1   +59.257, E3 +61065.191}
SPL {X  -159.990, Y  +624.023, Z    +0.000, E1   +69.513, E3 +61069.316}
SPL {X  -159.990, Y  +543.075, Z    +0.000, E1   +75.590, E3 +61092.964}
SPL {X  -156.121, Y  +342.530, Z    +0.000, E1   +75.868, E3 +61179.610}
SPL {X  -153.865, Y  +333.657, Z    +0.000, E1   +75.438, E3 +61189.215}
ENDSPLINE

SPLINE
SPL {X  -159.103, Y  +360.678, Z    +0.000, E1   +72.233, E3 +61207.318}
ENDSPLINE

SPLINE
SPL {X  -154.371, Y  +335.471, Z    +0.000, E1   +73.016, E3 +61215.889}
SPL {X  -148.318, Y  +317.512, Z    +0.000, E1   +73.488, E3 +61222.210}
SPL {X  -141.230, Y  +302.327, Z    +0.000, E1   +73.933, E3 +61226.764}
SPL {X  -135.697, Y  +292.747, Z    +0.000, E1   +74.259, E3 +61229.122}
SPL {X  -132.590, Y  +287.964, Z    +0.000, E1   +73.910, E3 +61234.150}
SPL {X  -129.541, Y  +283.606, Z    +0.000, E1   +73.551, E3 +61238.791}
SPL {X  -126.457, Y  +279.493, Z    +0.000, E1   +73.175, E3 +61243.190}
SPL {X  -122.770, Y  +274.912, Z    +0.000, E1   +72.712, E3 +61248.045}
SPL {X  -119.156, Y  +270.736, Z    +0.000, E1   +72.213, E3 +61252.394}
SPL {X  -117.531, Y  +268.949, Z    +0.000, E1   +71.964, E3 +61254.210}
SPL {X   -74.907, Y  +236.129, Z    +0.000, E1   +61.720, E3 +61331.246}
SPL {X   -72.759, Y  +235.012, Z    +0.000, E1   +56.036, E3 +61502.923}
ENDSPLINE

SPLINE
SPL {X  -110.316, Y  +261.624, Z    +0.000, E1   +58.739, E3 +61574.996}
SPL {X  -136.558, Y  +294.141, Z    +0.000, E1   +54.887, E3 +61596.793}
SPL {X  -153.807, Y  +333.452, Z    +0.000, E1   +40.945, E3 +61607.190}
SPL {X  -158.168, Y  +353.421, Z    +0.000, E1   +27.296, E3 +61609.584}
SPL {X  -159.556, Y  +365.719, Z    +0.000, E1   +15.845, E3 +61610.385}
SPL {X  -159.982, Y  +375.924, Z    +0.000, E1    +4.476, E3 +61610.686}
SPL {X  -159.990, Y  +379.800, Z    +0.000, E1    -0.377, E3 +61610.715}
SPL {X  -159.990, Y  +383.422, Z    +0.000, E1   -10.730, E3 +61610.758}
SPL {X  -159.990, Y  +387.978, Z    +0.000, E1   -23.882, E3 +61610.910}
SPL {X  -159.990, Y  +394.494, Z    +0.000, E1   -40.961, E3 +61611.291}
SPL {X  -159.990, Y  +400.492, Z    +0.000, E1   -51.837, E3 +61611.815}
SPL {X  -159.990, Y  +409.662, Z    +0.000, E1   -61.705, E3 +61612.926}
SPL {X  -159.990, Y  +434.697, Z    +0.000, E1   -71.504, E3 +61617.946}
SPL {X  -159.990, Y  +521.523, Z    +0.000, E1   -76.035, E3 +61644.227}
SPL {X  -154.459, Y  +718.205, Z    +0.000, E1   -76.329, E3 +61726.022}
SPL {X  -151.356, Y  +728.349, Z    +0.000, E1   -76.056, E3 +61734.238}
SPL {X  -147.124, Y  +739.360, Z    +0.000, E1   -75.690, E3 +61743.834}
SPL {X  -142.861, Y  +748.524, Z    +0.000, E1   -75.261, E3 +61752.519}
SPL {X  -138.117, Y  +757.250, Z    +0.000, E1   -74.803, E3 +61761.122}
SPL {X  -133.491, Y  +764.686, Z    +0.000, E1   -74.276, E3 +61768.863}
SPL {X  -130.530, Y  +769.013, Z    +0.000, E1   -73.929, E3 +61773.445}
SPL {X  -127.734, Y  +772.837, Z    +0.000, E1   -73.601, E3 +61777.497}
SPL {X  -124.765, Y  +776.652, Z    +0.000, E1   -73.233, E3 +61781.532}
SPL {X  -121.376, Y  +780.734, Z    +0.000, E1   -72.804, E3 +61785.793}
SPL {X  -118.281, Y  +784.233, Z    +0.000, E1   -72.371, E3 +61789.362}
SPL {X   -72.391, Y  +819.176, Z    +0.000, E1   -59.867, E3 +61885.247}
ENDSPLINE

SPLINE
SPL {X   -92.809, Y  +806.820, Z    +0.000, E1   -56.994, E3 +62078.043}
SPL {X  -120.521, Y  +781.721, Z    +0.000, E1   -56.766, E3 +62114.141}
SPL {X  -148.710, Y  +735.509, Z    +0.000, E1   -46.282, E3 +62135.422}
SPL {X  -157.559, Y  +704.285, Z    +0.000, E1   -29.037, E3 +62140.752}
SPL {X  -159.430, Y  +689.871, Z    +0.000, E1   -16.582, E3 +62141.902}
SPL {X  -159.960, Y  +679.609, Z    +0.000, E1    -6.021, E3 +62142.285}
SPL {X  -159.990, Y  +674.508, Z    +0.000, E1    -0.018, E3 +62142.344}
SPL {X  -159.990, Y  +672.787, Z    +0.000, E1    +4.022, E3 +62142.355}
SPL {X  -159.990, Y  +669.267, Z    +0.000, E1   +13.665, E3 +62142.426}
SPL {X  -159.990, Y  +665.069, Z    +0.000, E1   +25.376, E3 +62142.597}
SPL {X  -159.990, Y  +657.821, Z    +0.000, E1   +42.408, E3 +62143.100}
SPL {X  -159.990, Y  +645.368, Z    +0.000, E1   +59.257, E3 +62144.557}
SPL {X  -159.990, Y  +624.023, Z    +0.000, E1   +69.513, E3 +62148.681}
SPL {X  -159.990, Y  +543.075, Z    +0.000, E1   +75.590, E3 +62172.329}
SPL {X  -156.121, Y  +342.530, Z    +0.000, E1   +75.868, E3 +62258.976}
SPL {X  -153.498, Y  +332.386, Z    +0.000, E1   +75.628, E3 +62266.980}
ENDSPLINE

SPLINE
SPL {X  -155.252, Y  +338.851, Z    +0.000, E1   +74.632, E3 +62274.358}
SPL {X  -159.644, Y  +366.989, Z    +0.000, E1   +72.058, E3 +62284.106}
ENDSPLINE

SPLINE
SPL {X  -156.933, Y  +346.374, Z    +0.000, E1   +72.645, E3 +62291.996}
SPL {X  -151.144, Y  +325.039, Z    +0.000, E1   +73.323, E3 +62298.675}
SPL {X  -146.668, Y  +313.584, Z    +0.000, E1   +73.560, E3 +62303.157}
SPL {X  -141.230, Y  +302.327, Z    +0.000, E1   +73.933, E3 +62306.129}
SPL {X  -135.697, Y  +292.747, Z    +0.000, E1   +74.259, E3 +62308.487}
SPL {X  -132.590, Y  +287.964, Z    +0.000, E1   +73.910, E3 +62313.515}
SPL {X  -129.541, Y  +283.606, Z    +0.000, E1   +73.551, E3 +62318.156}
SPL {X  -126.457, Y  +279.493, Z    +0.000, E1   +73.175, E3 +62322.555}
SPL {X  -122.770, Y  +274.912, Z    +0.000, E1   +72.712, E3 +62327.410}
SPL {X  -118.941, Y  +270.496, Z    +0.000, E1   +72.188, E3 +62331.998}
SPL {X   -74.907, Y  +236.129, Z    +0.000, E1   +61.720, E3 +62410.611}
SPL {X   -72.759, Y  +235.012, Z    +0.000, E1   +56.036, E3 +62582.288}
ENDSPLINE

SPLINE
SPL {X  -123.257, Y  +275.497, Z    +0.000, E1   +57.800, E3 +62666.164}
SPL {X  -149.689, Y  +321.019, Z    +0.000, E1   +46.817, E3 +62684.265}
SPL {X  -157.484, Y  +349.293, Z    +0.000, E1   +30.654, E3 +62688.557}
SPL {X  -159.556, Y  +365.719, Z    +0.000, E1   +15.845, E3 +62689.750}
SPL {X  -159.982, Y  +375.924, Z    +0.000, E1    +4.476, E3 +62690.051}
SPL {X  -159.990, Y  +379.531, Z    +0.000, E1    -0.039, E3 +62690.078}
SPL {X  -159.990, Y  +382.420, Z    +0.000, E1    -7.600, E3 +62690.107}
SPL {X  -159.990, Y  +387.978, Z    +0.000, E1   -23.882, E3 +62690.275}
SPL {X  -159.990, Y  +396.850, Z    +0.000, E1   -45.459, E3 +62690.862}
SPL {X  -159.990, Y  +409.662, Z    +0.000, E1   -61.705, E3 +62692.291}
SPL {X  -159.990, Y  +434.697, Z    +0.000, E1   -71.504, E3 +62697.311}
SPL {X  -159.990, Y  +521.523, Z    +0.000, E1   -76.035, E3 +62723.592}
SPL {X  -154.459, Y  +718.205, Z    +0.000, E1   -76.329, E3 +62805.387}
SPL {X  -151.356, Y  +728.349, Z    +0.000, E1   -76.056, E3 +62813.603}
SPL {X  -148.399, Y  +736.287, Z    +0.000, E1   -75.788, E3 +62820.481}
SPL {X  -144.005, Y  +746.209, Z    +0.000, E1   -75.396, E3 +62829.597}
SPL {X  -138.117, Y  +757.250, Z    +0.000, E1   -74.803, E3 +62840.487}
SPL {X  -133.491, Y  +764.686, Z    +0.000, E1   -74.276, E3 +62848.228}
SPL {X  -128.839, Y  +771.354, Z    +0.000, E1   -73.759, E3 +62855.247}
SPL {X  -124.765, Y  +776.652, Z    +0.000, E1   -73.233, E3 +62860.897}
SPL {X  -121.376, Y  +780.734, Z    +0.000, E1   -72.804, E3 +62865.158}
SPL {X  -118.281, Y  +784.233, Z    +0.000, E1   -72.371, E3 +62868.727}
SPL {X   -72.391, Y  +819.176, Z    +0.000, E1   -59.867, E3 +62964.613}
ENDSPLINE

SPLINE
SPL {X  -116.241, Y  +786.431, Z    +0.000, E1   -57.120, E3 +63189.055}
SPL {X  -148.710, Y  +735.509, Z    +0.000, E1   -46.282, E3 +63214.787}
SPL {X  -157.559, Y  +704.285, Z    +0.000, E1   -29.037, E3 +63220.117}
SPL {X  -159.709, Y  +685.986, Z    +0.000, E1   -12.810, E3 +63221.449}
SPL {X  -159.990, Y  +674.648, Z    +0.000, E1    -0.349, E3 +63221.708}
SPL {X  -159.990, Y  +672.787, Z    +0.000, E1    +4.022, E3 +63221.720}
SPL {X  -159.990, Y  +669.267, Z    +0.000, E1   +13.665, E3 +63221.791}
SPL {X  -159.990, Y  +663.438, Z    +0.000, E1   +29.379, E3 +63222.061}
SPL {X  -159.990, Y  +655.264, Z    +0.000, E1   +47.291, E3 +63222.678}
SPL {X  -159.990, Y  +645.368, Z    +0.000, E1   +59.257, E3 +63223.922}
SPL {X  -159.990, Y  +624.023, Z    +0.000, E1   +69.513, E3 +63228.046}
SPL {X  -159.990, Y  +543.075, Z    +0.000, E1   +75.590, E3 +63251.694}
SPL {X  -156.121, Y  +342.530, Z    +0.000, E1   +75.868, E3 +63338.341}
SPL {X  -153.498, Y  +332.386, Z    +0.000, E1   +75.628, E3 +63346.345}
ENDSPLINE

SPLINE
SPL {X  -155.252, Y  +338.851, Z    +0.000, E1   +74.632, E3 +63353.723}
SPL {X  -159.103, Y  +360.678, Z    +0.000, E1   +72.233, E3 +63366.048}
ENDSPLINE

SPLINE
SPL {X  -154.371, Y  +335.471, Z    +0.000, E1   +73.016, E3 +63374.619}
SPL {X  -149.938, Y  +321.685, Z    +0.000, E1   +73.398, E3 +63379.313}
SPL {X  -145.016, Y  +309.920, Z    +0.000, E1   +73.647, E3 +63383.834}
SPL {X  -136.944, Y  +294.777, Z    +0.000, E1   +74.219, E3 +63387.136}
SPL {X  -132.590, Y  +287.964, Z    +0.000, E1   +73.910, E3 +63392.880}
SPL {X  -129.541, Y  +283.606, Z    +0.000, E1   +73.551, E3 +63397.521}
SPL {X  -125.403, Y  +278.147, Z    +0.000, E1   +73.063, E3 +63403.328}
SPL {X  -121.908, Y  +273.889, Z    +0.000, E1   +72.578, E3 +63407.874}
SPL {X  -119.156, Y  +270.736, Z    +0.000, E1   +72.213, E3 +63411.124}
SPL {X  -117.531, Y  +268.949, Z    +0.000, E1   +71.964, E3 +63412.940}
SPL {X   -74.907, Y  +236.129, Z    +0.000, E1   +61.720, E3 +63489.976}
ENDSPLINE

SPLINE
SPL {X   -94.059, Y  +248.080, Z    +0.000, E1   +58.275, E3 +63711.669}
SPL {X  -130.769, Y  +285.325, Z    +0.000, E1   +56.495, E3 +63751.546}
SPL {X  -149.689, Y  +321.019, Z    +0.000, E1   +46.817, E3 +63763.630}
SPL {X  -157.484, Y  +349.293, Z    +0.000, E1   +30.654, E3 +63767.922}
SPL {X  -159.556, Y  +365.719, Z    +0.000, E1   +15.845, E3 +63769.115}
SPL {X  -159.982, Y  +375.924, Z    +0.000, E1    +4.476, E3 +63769.417}
SPL {X  -159.990, Y  +379.531, Z    +0.000, E1    -0.039, E3 +63769.444}
SPL {X  -159.990, Y  +382.420, Z    +0.000, E1    -7.600, E3 +63769.472}
SPL {X  -159.990, Y  +386.504, Z    +0.000, E1   -19.860, E3 +63769.577}
SPL {X  -159.990, Y  +392.530, Z    +0.000, E1   -36.133, E3 +63769.893}
SPL {X  -159.990, Y  +400.492, Z    +0.000, E1   -51.837, E3 +63770.545}
SPL {X  -159.990, Y  +409.662, Z    +0.000, E1   -61.705, E3 +63771.656}
SPL {X  -159.990, Y  +434.697, Z    +0.000, E1   -71.504, E3 +63776.676}
SPL {X  -159.990, Y  +521.523, Z    +0.000, E1   -76.035, E3 +63802.957}
SPL {X  -154.459, Y  +718.205, Z    +0.000, E1   -76.329, E3 +63884.752}
SPL {X  -151.356, Y  +728.349, Z    +0.000, E1   -76.056, E3 +63892.968}
SPL {X  -148.399, Y  +736.287, Z    +0.000, E1   -75.788, E3 +63899.846}
SPL {X  -144.005, Y  +746.209, Z    +0.000, E1   -75.396, E3 +63908.962}
SPL {X  -138.117, Y  +757.250, Z    +0.000, E1   -74.803, E3 +63919.853}
SPL {X  -133.491, Y  +764.686, Z    +0.000, E1   -74.276, E3 +63927.593}
SPL {X  -128.839, Y  +771.354, Z    +0.000, E1   -73.759, E3 +63934.612}
SPL {X  -123.568, Y  +778.125, Z    +0.000, E1   -73.105, E3 +63941.784}
SPL {X  -118.985, Y  +783.455, Z    +0.000, E1   -72.490, E3 +63947.291}
SPL {X   -72.391, Y  +819.176, Z    +0.000, E1   -59.867, E3 +64043.978}
ENDSPLINE

SPLINE
SPL {X   -92.809, Y  +806.820, Z    +0.000, E1   -56.994, E3 +64236.773}
SPL {X  -120.521, Y  +781.721, Z    +0.000, E1   -56.766, E3 +64272.872}
SPL {X  -143.482, Y  +747.279, Z    +0.000, E1   -50.227, E3 +64290.884}
SPL {X  -154.118, Y  +719.449, Z    +0.000, E1   -38.836, E3 +64297.464}
SPL {X  -158.958, Y  +694.646, Z    +0.000, E1   -21.132, E3 +64300.315}
SPL {X  -159.960, Y  +679.609, Z    +0.000, E1    -6.021, E3 +64301.015}
SPL {X  -159.990, Y  +674.508, Z    +0.000, E1    -0.018, E3 +64301.074}
SPL {X  -159.990, Y  +672.787, Z    +0.000, E1    +4.022, E3 +64301.086}
SPL {X  -159.990, Y  +669.267, Z    +0.000, E1   +13.665, E3 +64301.156}
SPL {X  -159.990, Y  +663.438, Z    +0.000, E1   +29.379, E3 +64301.426}
SPL {X  -159.990, Y  +655.264, Z    +0.000, E1   +47.291, E3 +64302.043}
SPL {X  -159.990, Y  +645.368, Z    +0.000, E1   +59.257, E3 +64303.287}
SPL {X  -159.990, Y  +624.023, Z    +0.000, E1   +69.513, E3 +64307.412}
SPL {X  -159.990, Y  +543.075, Z    +0.000, E1   +75.590, E3 +64331.059}
SPL {X  -156.121, Y  +342.530, Z    +0.000, E1   +75.868, E3 +64417.706}
SPL {X  -153.498, Y  +332.386, Z    +0.000, E1   +75.628, E3 +64425.710}
ENDSPLINE

SPLINE
SPL {X  -155.252, Y  +338.851, Z    +0.000, E1   +74.632, E3 +64433.089}
SPL {X  -159.103, Y  +360.678, Z    +0.000, E1   +72.233, E3 +64445.413}
ENDSPLINE

SPLINE
SPL {X  -154.371, Y  +335.471, Z    +0.000, E1   +73.016, E3 +64453.984}
SPL {X  -149.938, Y  +321.685, Z    +0.000, E1   +73.398, E3 +64458.679}
SPL {X  -145.016, Y  +309.920, Z    +0.000, E1   +73.647, E3 +64463.199}
SPL {X  -139.138, Y  +298.522, Z    +0.000, E1   +74.138, E3 +64465.215}
SPL {X  -135.697, Y  +292.747, Z    +0.000, E1   +74.259, E3 +64467.217}
SPL {X  -132.590, Y  +287.964, Z    +0.000, E1   +73.910, E3 +64472.245}
SPL {X  -129.541, Y  +283.606, Z    +0.000, E1   +73.551, E3 +64476.886}
SPL {X  -126.457, Y  +279.493, Z    +0.000, E1   +73.175, E3 +64481.285}
SPL {X  -122.770, Y  +274.912, Z    +0.000, E1   +72.712, E3 +64486.140}
SPL {X  -118.941, Y  +270.496, Z    +0.000, E1   +72.188, E3 +64490.728}
SPL {X   -74.907, Y  +236.129, Z    +0.000, E1   +61.720, E3 +64569.341}
ENDSPLINE

SPLINE
SPL {X   -94.059, Y  +248.080, Z    +0.000, E1   +58.275, E3 +64791.034}
SPL {X  -136.558, Y  +294.141, Z    +0.000, E1   +54.887, E3 +64834.888}
SPL {X  -151.843, Y  +327.098, Z    +0.000, E1   +44.118, E3 +64844.248}
SPL {X  -157.484, Y  +349.293, Z    +0.000, E1   +30.654, E3 +64847.287}
SPL {X  -159.556, Y  +365.719, Z    +0.000, E1   +15.845, E3 +64848.480}
SPL {X  -159.982, Y  +375.924, Z    +0.000, E1    +4.476, E3 +64848.782}
SPL {X  -159.990, Y  +379.531, Z    +0.000, E1    -0.039, E3 +64848.809}
SPL {X  -159.990, Y  +382.420, Z    +0.000, E1    -7.600, E3 +64848.837}
SPL {X  -159.990, Y  +386.504, Z    +0.000, E1   -19.860, E3 +64848.942}
SPL {X  -159.990, Y  +392.530, Z    +0.000, E1   -36.133, E3 +64849.258}
SPL {X  -159.990, Y  +400.492, Z    +0.000, E1   -51.837, E3 +64849.910}
SPL {X  -159.990, Y  +409.662, Z    +0.000, E1   -61.705, E3 +64851.022}
SPL {X  -159.990, Y  +434.697, Z    +0.000, E1   -71.504, E3 +64856.042}
SPL {X  -159.990, Y  +521.523, Z    +0.000, E1   -76.035, E3 +64882.322}
SPL {X  -154.459, Y  +718.205, Z    +0.000, E1   -76.329, E3 +64964.117}
SPL {X  -151.356, Y  +728.349, Z    +0.000, E1   -76.056, E3 +64972.333}
SPL {X  -148.399, Y  +736.287, Z    +0.000, E1   -75.788, E3 +64979.212}
SPL {X  -144.005, Y  +746.209, Z    +0.000, E1   -75.396, E3 +64988.328}
SPL {X  -138.117, Y  +757.250, Z    +0.000, E1   -74.803, E3 +64999.218}
SPL {X  -133.491, Y  +764.686, Z    +0.000, E1   -74.276, E3 +65006.959}
SPL {X  -130.530, Y  +769.013, Z    +0.000, E1   -73.929, E3 +65011.540}
SPL {X  -127.734, Y  +772.837, Z    +0.000, E1   -73.601, E3 +65015.593}
SPL {X  -124.765, Y  +776.652, Z    +0.000, E1   -73.233, E3 +65019.627}
SPL {X  -121.376, Y  +780.734, Z    +0.000, E1   -72.804, E3 +65023.888}
SPL {X  -118.281, Y  +784.233, Z    +0.000, E1   -72.371, E3 +65027.457}
SPL {X   -72.391, Y  +819.176, Z    +0.000, E1   -59.867, E3 +65123.343}
ENDSPLINE

SPLINE
SPL {X   -92.809, Y  +806.820, Z    +0.000, E1   -56.994, E3 +65316.138}
SPL {X  -120.521, Y  +781.721, Z    +0.000, E1   -56.766, E3 +65352.237}
SPL {X  -143.482, Y  +747.279, Z    +0.000, E1   -50.227, E3 +65370.250}
SPL {X  -154.118, Y  +719.449, Z    +0.000, E1   -38.836, E3 +65376.829}
SPL {X  -158.958, Y  +694.646, Z    +0.000, E1   -21.132, E3 +65379.680}
SPL {X  -159.960, Y  +679.609, Z    +0.000, E1    -6.021, E3 +65380.380}
SPL {X  -159.990, Y  +674.508, Z    +0.000, E1    -0.018, E3 +65380.439}
SPL {X  -159.990, Y  +672.787, Z    +0.000, E1    +4.022, E3 +65380.451}
SPL {X  -159.990, Y  +669.267, Z    +0.000, E1   +13.665, E3 +65380.521}
SPL {X  -159.990, Y  +665.069, Z    +0.000, E1   +25.376, E3 +65380.693}
SPL {X  -159.990, Y  +657.821, Z    +0.000, E1   +42.408, E3 +65381.195}
SPL {X  -159.990, Y  +645.368, Z    +0.000, E1   +59.257, E3 +65382.652}
SPL {X  -159.990, Y  +624.023, Z    +0.000, E1   +69.513, E3 +65386.777}
SPL {X  -159.990, Y  +543.075, Z    +0.000, E1   +75.590, E3 +65410.425}
SPL {X  -156.121, Y  +342.530, Z    +0.000, E1   +75.868, E3 +65497.071}
SPL {X  -153.865, Y  +333.657, Z    +0.000, E1   +75.438, E3 +65506.675}
ENDSPLINE

SPLINE
SPL {X  -159.103, Y  +360.678, Z    +0.000, E1   +72.233, E3 +65524.778}
ENDSPLINE

SPLINE
SPL {X  -154.371, Y  +335.471, Z    +0.000, E1   +73.016, E3 +65533.349}
SPL {X  -148.318, Y  +317.512, Z    +0.000, E1   +73.488, E3 +65539.671}
SPL {X  -141.230, Y  +302.327, Z    +0.000, E1   +73.933, E3 +65544.224}
SPL {X  -135.697, Y  +292.747, Z    +0.000, E1   +74.259, E3 +65546.582}
SPL {X  -132.590, Y  +287.964, Z    +0.000, E1   +73.910, E3 +65551.610}
SPL {X  -129.541, Y  +283.606, Z    +0.000, E1   +73.551, E3 +65556.251}
SPL {X  -126.457, Y  +279.493, Z    +0.000, E1   +73.175, E3 +65560.650}
SPL {X  -122.770, Y  +274.912, Z    +0.000, E1   +72.712, E3 +65565.505}
SPL {X  -119.156, Y  +270.736, Z    +0.000, E1   +72.213, E3 +65569.855}
SPL {X  -117.531, Y  +268.949, Z    +0.000, E1   +71.964, E3 +65571.670}
SPL {X   -74.907, Y  +236.129, Z    +0.000, E1   +61.720, E3 +65648.706}
SPL {X   -72.759, Y  +235.012, Z    +0.000, E1   +56.036, E3 +65820.384}
ENDSPLINE

SPLINE
SPL {X  -110.316, Y  +261.624, Z    +0.000, E1   +58.739, E3 +65892.456}
SPL {X  -136.558, Y  +294.141, Z    +0.000, E1   +54.887, E3 +65914.253}
SPL {X  -153.807, Y  +333.452, Z    +0.000, E1   +40.945, E3 +65924.650}
SPL {X  -158.168, Y  +353.421, Z    +0.000, E1   +27.296, E3 +65927.044}
SPL {X  -159.556, Y  +365.719, Z    +0.000, E1   +15.845, E3 +65927.845}
SPL {X  -159.982, Y  +375.924, Z    +0.000, E1    +4.476, E3 +65928.147}
SPL {X  -159.990, Y  +379.800, Z    +0.000, E1    -0.377, E3 +65928.175}
SPL {X  -159.990, Y  +383.422, Z    +0.000, E1   -10.730, E3 +65928.218}
SPL {X  -159.990, Y  +387.978, Z    +0.000, E1   -23.882, E3 +65928.370}
SPL {X  -159.990, Y  +394.494, Z    +0.000, E1   -40.961, E3 +65928.751}
SPL {X  -159.990, Y  +400.492, Z    +0.000, E1   -51.837, E3 +65929.275}
SPL {X  -159.990, Y  +409.662, Z    +0.000, E1   -61.705, E3 +65930.387}
SPL {X  -159.990, Y  +434.697, Z    +0.000, E1   -71.504, E3 +65935.407}
SPL {X  -159.990, Y  +521.523, Z    +0.000, E1   -76.035, E3 +65961.687}
SPL {X  -154.459, Y  +718.205, Z    +0.000, E1   -76.329, E3 +66043.483}
SPL {X  -151.356, Y  +728.349, Z    +0.000, E1   -76.056, E3 +66051.698}
SPL {X  -147.124, Y  +739.360, Z    +0.000, E1   -75.690, E3 +66061.294}
SPL {X  -142.861, Y  +748.524, Z    +0.000, E1   -75.261, E3 +66069.979}
SPL {X  -138.117, Y  +757.250, Z    +0.000, E1   -74.803, E3 +66078.583}
SPL {X  -133.491, Y  +764.686, Z    +0.000, E1   -74.276, E3 +66086.324}
SPL {X  -130.530, Y  +769.013, Z    +0.000, E1   -73.929, E3 +66090.905}
SPL {X  -127.734, Y  +772.837, Z    +0.000, E1   -73.601, E3 +66094.958}
SPL {X  -124.765, Y  +776.652, Z    +0.000, E1   -73.233, E3 +66098.992}
SPL {X  -121.376, Y  +780.734, Z    +0.000, E1   -72.804, E3 +66103.254}
SPL {X  -118.281, Y  +784.233, Z    +0.000, E1   -72.371, E3 +66106.822}
SPL {X   -72.391, Y  +819.176, Z    +0.000, E1   -59.867, E3 +66202.708}
ENDSPLINE

SPLINE
SPL {X   -92.809, Y  +806.820, Z    +0.000, E1   -56.994, E3 +66395.503}
SPL {X  -120.521, Y  +781.721, Z    +0.000, E1   -56.766, E3 +66431.602}
SPL {X  -143.482, Y  +747.279, Z    +0.000, E1   -50.227, E3 +66449.615}
SPL {X  -154.118, Y  +719.449, Z    +0.000, E1   -38.836, E3 +66456.194}
SPL {X  -158.958, Y  +694.646, Z    +0.000, E1   -21.132, E3 +66459.045}
SPL {X  -159.960, Y  +679.609, Z    +0.000, E1    -6.021, E3 +66459.745}
SPL {X  -159.990, Y  +674.508, Z    +0.000, E1    -0.018, E3 +66459.804}
SPL {X  -159.990, Y  +672.787, Z    +0.000, E1    +4.022, E3 +66459.816}
SPL {X  -159.990, Y  +669.267, Z    +0.000, E1   +13.665, E3 +66459.886}
SPL {X  -159.990, Y  +665.069, Z    +0.000, E1   +25.376, E3 +66460.058}
SPL {X  -159.990, Y  +657.821, Z    +0.000, E1   +42.408, E3 +66460.560}
SPL {X  -159.990, Y  +645.368, Z    +0.000, E1   +59.257, E3 +66462.017}
SPL {X  -159.990, Y  +624.023, Z    +0.000, E1   +69.513, E3 +66466.142}
SPL {X  -159.990, Y  +543.075, Z    +0.000, E1   +75.590, E3 +66489.790}
SPL {X  -156.121, Y  +342.530, Z    +0.000, E1   +75.868, E3 +66576.436}
SPL {X  -153.865, Y  +333.657, Z    +0.000, E1   +75.438, E3 +66586.040}
ENDSPLINE

SPLINE
SPL {X  -159.103, Y  +360.678, Z    +0.000, E1   +72.233, E3 +66604.144}
ENDSPLINE

SPLINE
SPL {X  -154.371, Y  +335.471, Z    +0.000, E1   +73.016, E3 +66612.714}
SPL {X  -148.318, Y  +317.512, Z    +0.000, E1   +73.488, E3 +66619.036}
SPL {X  -141.230, Y  +302.327, Z    +0.000, E1   +73.933, E3 +66623.589}
SPL {X  -135.697, Y  +292.747, Z    +0.000, E1   +74.259, E3 +66625.947}
SPL {X  -132.590, Y  +287.964, Z    +0.000, E1   +73.910, E3 +66630.976}
SPL {X  -129.541, Y  +283.606, Z    +0.000, E1   +73.551, E3 +66635.616}
SPL {X  -126.457, Y  +279.493, Z    +0.000, E1   +73.175, E3 +66640.015}
SPL {X  -122.770, Y  +274.912, Z    +0.000, E1   +72.712, E3 +66644.870}
SPL {X  -119.156, Y  +270.736, Z    +0.000, E1   +72.213, E3 +66649.220}
SPL {X  -117.531, Y  +268.949, Z    +0.000, E1   +71.964, E3 +66651.035}
SPL {X   -74.907, Y  +236.129, Z    +0.000, E1   +61.720, E3 +66728.071}
SPL {X   -72.759, Y  +235.012, Z    +0.000, E1   +56.036, E3 +66899.749}
ENDSPLINE

SPLINE
SPL {X  -110.316, Y  +261.624, Z    +0.000, E1   +58.739, E3 +66971.821}
SPL {X  -136.558, Y  +294.141, Z    +0.000, E1   +54.887, E3 +66993.618}
SPL {X  -153.807, Y  +333.452, Z    +0.000, E1   +40.945, E3 +67004.015}
SPL {X  -158.168, Y  +353.421, Z    +0.000, E1   +27.296, E3 +67006.409}
SPL {X  -159.556, Y  +365.719, Z    +0.000, E1   +15.845, E3 +67007.210}
SPL {X  -159.982, Y  +375.924, Z    +0.000, E1    +4.476, E3 +67007.512}
SPL {X  -159.990, Y  +379.800, Z    +0.000, E1    -0.377, E3 +67007.540}
SPL {X  -159.990, Y  +383.422, Z    +0.000, E1   -10.730, E3 +67007.583}
SPL {X  -159.990, Y  +387.978, Z    +0.000, E1   -23.882, E3 +67007.736}
SPL {X  -159.990, Y  +394.494, Z    +0.000, E1   -40.961, E3 +67008.116}
SPL {X  -159.990, Y  +400.492, Z    +0.000, E1   -51.837, E3 +67008.641}
SPL {X  -159.990, Y  +409.662, Z    +0.000, E1   -61.705, E3 +67009.752}
SPL {X  -159.990, Y  +434.697, Z    +0.000, E1   -71.504, E3 +67014.772}
SPL {X  -159.990, Y  +521.523, Z    +0.000, E1   -76.035, E3 +67041.052}
SPL {X  -154.459, Y  +718.205, Z    +0.000, E1   -76.329, E3 +67122.848}
SPL {X  -151.356, Y  +728.349, Z    +0.000, E1   -76.056, E3 +67131.063}
SPL {X  -147.124, Y  +739.360, Z    +0.000, E1   -75.690, E3 +67140.659}
SPL {X  -142.861, Y  +748.524, Z    +0.000, E1   -75.261, E3 +67149.344}
SPL {X  -138.117, Y  +757.250, Z    +0.000, E1   -74.803, E3 +67157.948}
SPL {X  -133.491, Y  +764.686, Z    +0.000, E1   -74.276, E3 +67165.689}
SPL {X  -130.530, Y  +769.013, Z    +0.000, E1   -73.929, E3 +67170.271}
SPL {X  -127.734, Y  +772.837, Z    +0.000, E1   -73.601, E3 +67174.323}
SPL {X  -124.765, Y  +776.652, Z    +0.000, E1   -73.233, E3 +67178.357}
SPL {X  -121.376, Y  +780.734, Z    +0.000, E1   -72.804, E3 +67182.619}
SPL {X  -118.281, Y  +784.233, Z    +0.000, E1   -72.371, E3 +67186.187}
SPL {X   -72.391, Y  +819.176, Z    +0.000, E1   -59.867, E3 +67282.073}
ENDSPLINE

SPLINE
SPL {X   -92.809, Y  +806.820, Z    +0.000, E1   -56.994, E3 +67474.868}
SPL {X  -120.521, Y  +781.721, Z    +0.000, E1   -56.766, E3 +67510.967}
SPL {X  -143.482, Y  +747.279, Z    +0.000, E1   -50.227, E3 +67528.980}
SPL {X  -154.118, Y  +719.449, Z    +0.000, E1   -38.836, E3 +67535.559}
SPL {X  -158.958, Y  +694.646, Z    +0.000, E1   -21.132, E3 +67538.410}
SPL {X  -159.960, Y  +679.609, Z    +0.000, E1    -6.021, E3 +67539.110}
SPL {X  -159.990, Y  +674.508, Z    +0.000, E1    -0.018, E3 +67539.169}
SPL {X  -159.990, Y  +672.787, Z    +0.000, E1    +4.022, E3 +67539.181}
SPL {X  -159.990, Y  +669.267, Z    +0.000, E1   +13.665, E3 +67539.251}
SPL {X  -159.990, Y  +665.069, Z    +0.000, E1   +25.376, E3 +67539.423}
SPL {X  -159.990, Y  +657.821, Z    +0.000, E1   +42.408, E3 +67539.925}
SPL {X  -159.990, Y  +645.368, Z    +0.000, E1   +59.257, E3 +67541.382}
SPL {X  -159.990, Y  +624.023, Z    +0.000, E1   +69.513, E3 +67545.507}
SPL {X  -159.990, Y  +543.075, Z    +0.000, E1   +75.590, E3 +67569.155}
SPL {X  -156.121, Y  +342.530, Z    +0.000, E1   +75.868, E3 +67655.801}
SPL {X  -153.865, Y  +333.657, Z    +0.000, E1   +75.438, E3 +67665.405}
ENDSPLINE

SPLINE
SPL {X  -159.103, Y  +360.678, Z    +0.000, E1   +72.233, E3 +67683.509}
ENDSPLINE

SPLINE
SPL {X  -154.371, Y  +335.471, Z    +0.000, E1   +73.016, E3 +67692.079}
SPL {X  -148.318, Y  +317.512, Z    +0.000, E1   +73.488, E3 +67698.401}
SPL {X  -141.226, Y  +302.320, Z    +0.000, E1   +73.932, E3 +67702.964}
SPL {X  -140.628, Y  +301.207, Z    +0.000, E1   +72.742, E3 +67713.253}
SPL {X  -137.438, Y  +295.601, Z    +0.000, E1   +72.365, E3 +67719.359}
SPL {X  -134.156, Y  +290.328, Z    +0.000, E1   +71.962, E3 +67725.230}
SPL {X  -130.677, Y  +285.194, Z    +0.000, E1   +71.519, E3 +67731.035}
SPL {X  -127.147, Y  +280.390, Z    +0.000, E1   +71.042, E3 +67736.519}
SPL {X  -123.431, Y  +275.709, Z    +0.000, E1   +70.518, E3 +67741.842}
SPL {X  -120.392, Y  +272.131, Z    +0.000, E1   +70.053, E3 +67745.862}
SPL {X   -79.311, Y  +238.552, Z    +0.000, E1   +58.563, E3 +67841.101}
ENDSPLINE

SPLINE
SPL {X  -105.077, Y  +256.854, Z    +0.000, E1   +55.187, E3 +68028.654}
SPL {X  -133.208, Y  +288.886, Z    +0.000, E1   +52.003, E3 +68061.755}
SPL {X  -149.825, Y  +321.381, Z    +0.000, E1   +42.580, E3 +68074.908}
SPL {X  -156.491, Y  +344.222, Z    +0.000, E1   +30.612, E3 +68079.414}
SPL {X  -159.275, Y  +362.387, Z    +0.000, E1   +16.907, E3 +68081.328}
SPL {X  -159.964, Y  +374.630, Z    +0.000, E1    +5.249, E3 +68081.902}
SPL {X  -159.990, Y  +379.735, Z    +0.000, E1    -0.236, E3 +68081.959}
SPL {X  -159.990, Y  +382.878, Z    +0.000, E1    -7.664, E3 +68081.998}
SPL {X  -159.990, Y  +387.459, Z    +0.000, E1   -18.927, E3 +68082.175}
SPL {X  -159.990, Y  +395.361, Z    +0.000, E1   -37.740, E3 +68082.739}
SPL {X  -159.990, Y  +406.369, Z    +0.000, E1   -54.148, E3 +68084.145}
SPL {X  -159.990, Y  +426.617, Z    +0.000, E1   -66.230, E3 +68088.394}
SPL {X  -159.990, Y  +499.521, Z    +0.000, E1   -73.662, E3 +68111.721}
SPL {X  -159.629, Y  +687.249, Z    +0.000, E1   -74.539, E3 +68199.605}
SPL {X  -157.983, Y  +701.765, Z    +0.000, E1   -74.384, E3 +68209.837}
SPL {X  -155.520, Y  +714.054, Z    +0.000, E1   -74.151, E3 +68219.591}
SPL {X  -152.569, Y  +724.660, Z    +0.000, E1   -73.857, E3 +68228.826}
SPL {X  -149.625, Y  +733.149, Z    +0.000, E1   -73.553, E3 +68236.761}
SPL {X  -146.617, Y  +740.532, Z    +0.000, E1   -73.233, E3 +68244.038}
SPL {X  -143.394, Y  +747.457, Z    +0.000, E1   -72.883, E3 +68251.135}
SPL {X  -140.332, Y  +753.336, Z    +0.000, E1   -72.527, E3 +68257.410}
SPL {X  -137.187, Y  +758.820, Z    +0.000, E1   -72.156, E3 +68263.413}
SPL {X  -134.014, Y  +763.891, Z    +0.000, E1   -71.759, E3 +68269.098}
SPL {X  -130.657, Y  +768.834, Z    +0.000, E1   -71.330, E3 +68274.714}
SPL {X  -126.937, Y  +773.885, Z    +0.000, E1   -70.823, E3 +68280.515}
SPL {X  -122.983, Y  +778.833, Z    +0.000, E1   -70.262, E3 +68286.160}
SPL {X  -120.205, Y  +782.082, Z    +0.000, E1   -69.822, E3 +68289.828}
SPL {X   -77.717, Y  +816.346, Z    +0.000, E1   -57.422, E3 +68397.680}
SPL {X   -74.440, Y  +818.117, Z    +0.000, E1   -54.647, E3 +68450.919}
ENDSPLINE

SPLINE
SPL {X  -124.054, Y  +777.532, Z    +0.000, E1   -54.436, E3 +68598.995}
SPL {X  -149.719, Y  +732.901, Z    +0.000, E1   -43.150, E3 +68619.809}
SPL {X  -158.004, Y  +701.630, Z    +0.000, E1   -25.366, E3 +68625.274}
SPL {X  -159.639, Y  +687.095, Z    +0.000, E1   -12.931, E3 +68626.432}
SPL {X  -159.981, Y  +678.202, Z    +0.000, E1    -4.129, E3 +68626.726}
SPL {X  -159.990, Y  +674.500, Z    +0.000, E1    +0.000, E3 +68626.764}
SPL {X  -159.990, Y  +672.677, Z    +0.000, E1    +3.879, E3 +68626.779}
SPL {X  -159.990, Y  +669.117, Z    +0.000, E1   +12.900, E3 +68626.862}
SPL {X  -159.990, Y  +663.639, Z    +0.000, E1   +26.675, E3 +68627.147}
SPL {X  -159.990, Y  +656.057, Z    +0.000, E1   +43.288, E3 +68627.803}
SPL {X  -159.990, Y  +645.786, Z    +0.000, E1   +56.338, E3 +68629.294}
SPL {X  -159.990, Y  +623.264, Z    +0.000, E1   +67.753, E3 +68634.220}
SPL {X  -159.990, Y  +547.268, Z    +0.000, E1   +73.735, E3 +68659.908}
SPL {X  -159.091, Y  +360.560, Z    +0.000, E1   +74.726, E3 +68746.235}
SPL {X  -156.418, Y  +343.879, Z    +0.000, E1   +74.473, E3 +68758.660}
SPL {X  -153.414, Y  +332.103, Z    +0.000, E1   +74.378, E3 +68766.335}
SPL {X  -141.909, Y  +303.617, Z    +0.000, E1   +76.515, E3 +68758.865}
ENDSPLINE

SPLINE
SPL {X  -142.567, Y  +304.895, Z    +0.000, E1   +75.566, E3 +68767.680}
ENDSPLINE

SPLINE
SPL {X  -141.999, Y  +303.790, Z    +0.000, E1   +74.633, E3 +68776.931}
SPL {X  -141.780, Y  +303.371, Z    +0.000, E1   +73.549, E3 +68786.505}
SPL {X  -140.619, Y  +301.190, Z    +0.000, E1   +72.741, E3 +68794.351}
SPL {X  -137.438, Y  +295.601, Z    +0.000, E1   +72.365, E3 +68800.440}
SPL {X  -134.156, Y  +290.328, Z    +0.000, E1   +71.962, E3 +68806.311}
SPL {X  -130.677, Y  +285.194, Z    +0.000, E1   +71.519, E3 +68812.116}
SPL {X  -127.147, Y  +280.390, Z    +0.000, E1   +71.042, E3 +68817.600}
SPL {X  -123.431, Y  +275.709, Z    +0.000, E1   +70.518, E3 +68822.923}
SPL {X  -120.392, Y  +272.131, Z    +0.000, E1   +70.053, E3 +68826.943}
SPL {X   -79.311, Y  +238.552, Z    +0.000, E1   +58.563, E3 +68922.182}
ENDSPLINE

SPLINE
SPL {X  -105.077, Y  +256.854, Z    +0.000, E1   +55.187, E3 +69109.735}
SPL {X  -133.208, Y  +288.886, Z    +0.000, E1   +52.003, E3 +69142.836}
SPL {X  -149.825, Y  +321.381, Z    +0.000, E1   +42.580, E3 +69155.989}
SPL {X  -157.376, Y  +348.695, Z    +0.000, E1   +27.651, E3 +69161.074}
SPL {X  -159.486, Y  +364.808, Z    +0.000, E1   +14.693, E3 +69162.577}
SPL {X  -159.964, Y  +374.630, Z    +0.000, E1    +5.249, E3 +69162.983}
SPL {X  -159.990, Y  +379.484, Z    +0.000, E1    +0.034, E3 +69163.038}
SPL {X  -159.990, Y  +381.639, Z    +0.000, E1    -4.454, E3 +69163.060}
SPL {X  -159.990, Y  +385.871, Z    +0.000, E1   -15.161, E3 +69163.176}
SPL {X  -159.990, Y  +391.065, Z    +0.000, E1   -28.187, E3 +69163.464}
SPL {X  -159.990, Y  +399.326, Z    +0.000, E1   -44.934, E3 +69164.247}
SPL {X  -159.990, Y  +408.817, Z    +0.000, E1   -56.572, E3 +69165.620}
SPL {X  -159.990, Y  +426.617, Z    +0.000, E1   -66.230, E3 +69169.475}
SPL {X  -159.990, Y  +499.521, Z    +0.000, E1   -73.662, E3 +69192.802}
SPL {X  -159.629, Y  +687.249, Z    +0.000, E1   -74.539, E3 +69280.686}
SPL {X  -157.983, Y  +701.765, Z    +0.000, E1   -74.384, E3 +69290.919}
SPL {X  -155.520, Y  +714.054, Z    +0.000, E1   -74.151, E3 +69300.673}
SPL {X  -152.569, Y  +724.660, Z    +0.000, E1   -73.857, E3 +69309.907}
SPL {X  -149.625, Y  +733.149, Z    +0.000, E1   -73.553, E3 +69317.842}
SPL {X  -146.617, Y  +740.532, Z    +0.000, E1   -73.233, E3 +69325.119}
SPL {X  -143.394, Y  +747.457, Z    +0.000, E1   -72.883, E3 +69332.216}
SPL {X  -140.332, Y  +753.336, Z    +0.000, E1   -72.527, E3 +69338.491}
SPL {X  -137.187, Y  +758.820, Z    +0.000, E1   -72.156, E3 +69344.494}
SPL {X  -134.014, Y  +763.891, Z    +0.000, E1   -71.759, E3 +69350.179}
SPL {X  -129.643, Y  +770.252, Z    +0.000, E1   -71.218, E3 +69357.386}
SPL {X  -125.230, Y  +776.071, Z    +0.000, E1   -70.580, E3 +69364.104}
SPL {X  -122.263, Y  +779.692, Z    +0.000, E1   -70.136, E3 +69368.234}
SPL {X  -120.205, Y  +782.082, Z    +0.000, E1   -69.822, E3 +69370.909}
SPL {X   -75.772, Y  +817.409, Z    +0.000, E1   -56.226, E3 +69496.848}
ENDSPLINE

SPLINE
SPL {X  -124.054, Y  +777.532, Z    +0.000, E1   -54.436, E3 +69680.076}
SPL {X  -145.922, Y  +742.101, Z    +0.000, E1   -46.535, E3 +69698.346}
SPL {X  -155.216, Y  +715.293, Z    +0.000, E1   -34.460, E3 +69704.538}
SPL {X  -158.715, Y  +696.660, Z    +0.000, E1   -21.368, E3 +69706.866}
SPL {X  -159.639, Y  +687.095, Z    +0.000, E1   -12.931, E3 +69707.513}
SPL {X  -159.981, Y  +678.202, Z    +0.000, E1    -4.129, E3 +69707.807}
SPL {X  -159.990, Y  +674.500, Z    +0.000, E1    +0.000, E3 +69707.845}
SPL {X  -159.990, Y  +672.677, Z    +0.000, E1    +3.879, E3 +69707.860}
SPL {X  -159.990, Y  +669.117, Z    +0.000, E1   +12.900, E3 +69707.943}
SPL {X  -159.990, Y  +663.639, Z    +0.000, E1   +26.675, E3 +69708.228}
SPL {X  -159.990, Y  +656.057, Z    +0.000, E1   +43.288, E3 +69708.884}
SPL {X  -159.990, Y  +647.797, Z    +0.000, E1   +54.469, E3 +69710.021}
SPL {X  -159.990, Y  +630.178, Z    +0.000, E1   +65.480, E3 +69713.705}
SPL {X  -159.990, Y  +547.268, Z    +0.000, E1   +73.735, E3 +69740.989}
SPL {X  -159.626, Y  +366.721, Z    +0.000, E1   +74.756, E3 +69823.255}
SPL {X  -158.582, Y  +356.317, Z    +0.000, E1   +74.662, E3 +69830.348}
SPL {X  -156.418, Y  +343.879, Z    +0.000, E1   +74.473, E3 +69839.741}
SPL {X  -153.414, Y  +332.103, Z    +0.000, E1   +74.378, E3 +69847.416}
SPL {X  -141.909, Y  +303.617, Z    +0.000, E1   +76.515, E3 +69839.946}
ENDSPLINE

SPLINE
SPL {X  -142.567, Y  +304.895, Z    +0.000, E1   +75.566, E3 +69848.761}
ENDSPLINE

SPLINE
SPL {X  -141.999, Y  +303.790, Z    +0.000, E1   +74.633, E3 +69858.012}
SPL {X  -141.780, Y  +303.371, Z    +0.000, E1   +73.549, E3 +69867.586}
SPL {X  -140.619, Y  +301.190, Z    +0.000, E1   +72.741, E3 +69875.433}
SPL {X  -137.438, Y  +295.601, Z    +0.000, E1   +72.365, E3 +69881.521}
SPL {X  -134.156, Y  +290.328, Z    +0.000, E1   +71.962, E3 +69887.392}
SPL {X  -130.677, Y  +285.194, Z    +0.000, E1   +71.519, E3 +69893.197}
SPL {X  -127.147, Y  +280.390, Z    +0.000, E1   +71.042, E3 +69898.681}
SPL {X  -123.431, Y  +275.709, Z    +0.000, E1   +70.518, E3 +69904.004}
SPL {X  -120.392, Y  +272.131, Z    +0.000, E1   +70.053, E3 +69908.024}
SPL {X   -79.311, Y  +238.552, Z    +0.000, E1   +58.563, E3 +70003.263}
ENDSPLINE

SPLINE
SPL {X  -105.077, Y  +256.854, Z    +0.000, E1   +55.187, E3 +70190.816}
SPL {X  -133.208, Y  +288.886, Z    +0.000, E1   +52.003, E3 +70223.917}
SPL {X  -149.825, Y  +321.381, Z    +0.000, E1   +42.580, E3 +70237.070}
SPL {X  -157.376, Y  +348.695, Z    +0.000, E1   +27.651, E3 +70242.155}
SPL {X  -159.486, Y  +364.808, Z    +0.000, E1   +14.693, E3 +70243.659}
SPL {X  -159.964, Y  +374.630, Z    +0.000, E1    +5.249, E3 +70244.064}
SPL {X  -159.990, Y  +379.484, Z    +0.000, E1    +0.034, E3 +70244.120}
SPL {X  -159.990, Y  +381.639, Z    +0.000, E1    -4.454, E3 +70244.141}
SPL {X  -159.990, Y  +385.871, Z    +0.000, E1   -15.161, E3 +70244.257}
SPL {X  -159.990, Y  +391.065, Z    +0.000, E1   -28.187, E3 +70244.545}
SPL {X  -159.990, Y  +399.326, Z    +0.000, E1   -44.934, E3 +70245.328}
SPL {X  -159.990, Y  +408.817, Z    +0.000, E1   -56.572, E3 +70246.701}
SPL {X  -159.990, Y  +426.617, Z    +0.000, E1   -66.230, E3 +70250.557}
SPL {X  -159.990, Y  +499.521, Z    +0.000, E1   -73.662, E3 +70273.883}
SPL {X  -159.629, Y  +687.249, Z    +0.000, E1   -74.539, E3 +70361.767}
SPL {X  -157.983, Y  +701.765, Z    +0.000, E1   -74.384, E3 +70372.000}
SPL {X  -155.520, Y  +714.054, Z    +0.000, E1   -74.151, E3 +70381.754}
SPL {X  -152.569, Y  +724.660, Z    +0.000, E1   -73.857, E3 +70390.988}
SPL {X  -149.625, Y  +733.149, Z    +0.000, E1   -73.553, E3 +70398.923}
SPL {X  -146.617, Y  +740.532, Z    +0.000, E1   -73.233, E3 +70406.200}
SPL {X  -143.394, Y  +747.457, Z    +0.000, E1   -72.883, E3 +70413.297}
SPL {X  -140.332, Y  +753.336, Z    +0.000, E1   -72.527, E3 +70419.572}
SPL {X  -137.187, Y  +758.820, Z    +0.000, E1   -72.156, E3 +70425.575}
SPL {X  -134.014, Y  +763.891, Z    +0.000, E1   -71.759, E3 +70431.260}
SPL {X  -129.643, Y  +770.252, Z    +0.000, E1   -71.218, E3 +70438.467}
SPL {X  -125.230, Y  +776.071, Z    +0.000, E1   -70.580, E3 +70445.186}
SPL {X  -121.287, Y  +780.838, Z    +0.000, E1   -70.013, E3 +70450.577}
SPL {X   -75.772, Y  +817.409, Z    +0.000, E1   -56.226, E3 +70577.929}
ENDSPLINE

SPLINE
SPL {X  -124.054, Y  +777.532, Z    +0.000, E1   -54.436, E3 +70761.157}
SPL {X  -145.922, Y  +742.101, Z    +0.000, E1   -46.535, E3 +70779.427}
SPL {X  -155.216, Y  +715.293, Z    +0.000, E1   -34.460, E3 +70785.619}
SPL {X  -158.715, Y  +696.660, Z    +0.000, E1   -21.368, E3 +70787.947}
SPL {X  -159.838, Y  +683.473, Z    +0.000, E1    -9.532, E3 +70788.743}
SPL {X  -159.990, Y  +674.579, Z    +0.000, E1    -0.168, E3 +70788.925}
SPL {X  -159.990, Y  +672.677, Z    +0.000, E1    +3.879, E3 +70788.941}
SPL {X  -159.990, Y  +669.117, Z    +0.000, E1   +12.900, E3 +70789.024}
SPL {X  -159.990, Y  +663.639, Z    +0.000, E1   +26.675, E3 +70789.309}
SPL {X  -159.990, Y  +656.057, Z    +0.000, E1   +43.288, E3 +70789.965}
SPL {X  -159.990, Y  +647.797, Z    +0.000, E1   +54.469, E3 +70791.102}
SPL {X  -159.990, Y  +630.178, Z    +0.000, E1   +65.480, E3 +70794.786}
SPL {X  -159.990, Y  +547.268, Z    +0.000, E1   +73.735, E3 +70822.070}
SPL {X  -159.091, Y  +360.560, Z    +0.000, E1   +74.726, E3 +70908.397}
SPL {X  -156.418, Y  +343.879, Z    +0.000, E1   +74.473, E3 +70920.822}
SPL {X  -153.414, Y  +332.103, Z    +0.000, E1   +74.378, E3 +70928.497}
SPL {X  -141.909, Y  +303.617, Z    +0.000, E1   +76.515, E3 +70921.027}
ENDSPLINE

SPLINE
SPL {X  -142.567, Y  +304.895, Z    +0.000, E1   +75.566, E3 +70929.842}
ENDSPLINE

SPLINE
SPL {X  -141.999, Y  +303.790, Z    +0.000, E1   +74.633, E3 +70939.093}
SPL {X  -141.780, Y  +303.371, Z    +0.000, E1   +73.549, E3 +70948.667}
SPL {X  -140.619, Y  +301.190, Z    +0.000, E1   +72.741, E3 +70956.514}
SPL {X  -137.438, Y  +295.601, Z    +0.000, E1   +72.365, E3 +70962.602}
SPL {X  -134.156, Y  +290.328, Z    +0.000, E1   +71.962, E3 +70968.473}
SPL {X  -130.677, Y  +285.194, Z    +0.000, E1   +71.519, E3 +70974.278}
SPL {X  -127.147, Y  +280.390, Z    +0.000, E1   +71.042, E3 +70979.762}
SPL {X  -123.431, Y  +275.709, Z    +0.000, E1   +70.518, E3 +70985.085}
SPL {X  -120.392, Y  +272.131, Z    +0.000, E1   +70.053, E3 +70989.105}
SPL {X   -79.311, Y  +238.552, Z    +0.000, E1   +58.563, E3 +71084.344}
ENDSPLINE

SPLINE
SPL {X  -105.077, Y  +256.854, Z    +0.000, E1   +55.187, E3 +71271.897}
SPL {X  -133.208, Y  +288.886, Z    +0.000, E1   +52.003, E3 +71304.998}
SPL {X  -149.825, Y  +321.381, Z    +0.000, E1   +42.580, E3 +71318.151}
SPL {X  -157.376, Y  +348.695, Z    +0.000, E1   +27.651, E3 +71323.236}
SPL {X  -159.486, Y  +364.808, Z    +0.000, E1   +14.693, E3 +71324.740}
SPL {X  -159.964, Y  +374.630, Z    +0.000, E1    +5.249, E3 +71325.145}
SPL {X  -159.990, Y  +379.735, Z    +0.000, E1    -0.236, E3 +71325.202}
SPL {X  -159.990, Y  +384.648, Z    +0.000, E1   -11.739, E3 +71325.299}
SPL {X  -159.990, Y  +391.065, Z    +0.000, E1   -28.187, E3 +71325.626}
SPL {X  -159.990, Y  +397.286, Z    +0.000, E1   -41.591, E3 +71326.169}
SPL {X  -159.990, Y  +406.369, Z    +0.000, E1   -54.148, E3 +71327.388}
SPL {X  -159.990, Y  +426.617, Z    +0.000, E1   -66.230, E3 +71331.638}
SPL {X  -159.990, Y  +499.521, Z    +0.000, E1   -73.662, E3 +71354.964}
SPL {X  -159.629, Y  +687.249, Z    +0.000, E1   -74.539, E3 +71442.848}
SPL {X  -157.983, Y  +701.765, Z    +0.000, E1   -74.384, E3 +71453.081}
SPL {X  -155.520, Y  +714.054, Z    +0.000, E1   -74.151, E3 +71462.835}
SPL {X  -152.569, Y  +724.660, Z    +0.000, E1   -73.857, E3 +71472.069}
SPL {X  -149.625, Y  +733.149, Z    +0.000, E1   -73.553, E3 +71480.005}
SPL {X  -146.617, Y  +740.532, Z    +0.000, E1   -73.233, E3 +71487.281}
SPL {X  -143.394, Y  +747.457, Z    +0.000, E1   -72.883, E3 +71494.378}
SPL {X  -140.332, Y  +753.336, Z    +0.000, E1   -72.527, E3 +71500.653}
SPL {X  -137.187, Y  +758.820, Z    +0.000, E1   -72.156, E3 +71506.656}
SPL {X  -134.014, Y  +763.891, Z    +0.000, E1   -71.759, E3 +71512.341}
SPL {X  -130.657, Y  +768.834, Z    +0.000, E1   -71.330, E3 +71517.957}
SPL {X  -126.020, Y  +775.068, Z    +0.000, E1   -70.718, E3 +71525.084}
SPL {X  -121.287, Y  +780.838, Z    +0.000, E1   -70.013, E3 +71531.658}
SPL {X   -75.772, Y  +817.409, Z    +0.000, E1   -56.226, E3 +71659.010}
ENDSPLINE

SPLINE
SPL {X  -124.054, Y  +777.532, Z    +0.000, E1   -54.436, E3 +71842.238}
SPL {X  -149.719, Y  +732.901, Z    +0.000, E1   -43.150, E3 +71863.053}
SPL {X  -158.004, Y  +701.630, Z    +0.000, E1   -25.366, E3 +71868.517}
SPL {X  -159.639, Y  +687.095, Z    +0.000, E1   -12.931, E3 +71869.675}
SPL {X  -159.981, Y  +678.202, Z    +0.000, E1    -4.129, E3 +71869.969}
SPL {X  -159.990, Y  +674.500, Z    +0.000, E1    +0.000, E3 +71870.007}
SPL {X  -159.990, Y  +672.677, Z    +0.000, E1    +3.879, E3 +71870.022}
SPL {X  -159.990, Y  +669.117, Z    +0.000, E1   +12.900, E3 +71870.105}
SPL {X  -159.990, Y  +663.639, Z    +0.000, E1   +26.675, E3 +71870.390}
SPL {X  -159.990, Y  +656.057, Z    +0.000, E1   +43.288, E3 +71871.046}
SPL {X  -159.990, Y  +645.786, Z    +0.000, E1   +56.338, E3 +71872.538}
SPL {X  -159.990, Y  +623.264, Z    +0.000, E1   +67.753, E3 +71877.463}
SPL {X  -159.990, Y  +547.268, Z    +0.000, E1   +73.735, E3 +71903.151}
SPL {X  -159.091, Y  +360.560, Z    +0.000, E1   +74.726, E3 +71989.478}
SPL {X  -156.418, Y  +343.879, Z    +0.000, E1   +74.473, E3 +72001.903}
SPL {X  -153.414, Y  +332.103, Z    +0.000, E1   +74.378, E3 +72009.578}
SPL {X  -141.909, Y  +303.617, Z    +0.000, E1   +76.515, E3 +72002.108}
ENDSPLINE

SPLINE
SPL {X  -142.567, Y  +304.895, Z    +0.000, E1   +75.566, E3 +72010.923}
ENDSPLINE

SPLINE
SPL {X  -141.999, Y  +303.790, Z    +0.000, E1   +74.633, E3 +72020.174}
SPL {X  -141.780, Y  +303.371, Z    +0.000, E1   +73.549, E3 +72029.748}
SPL {X  -140.619, Y  +301.190, Z    +0.000, E1   +72.741, E3 +72037.595}
SPL {X  -137.438, Y  +295.601, Z    +0.000, E1   +72.365, E3 +72043.683}
SPL {X  -134.156, Y  +290.328, Z    +0.000, E1   +71.962, E3 +72049.554}
SPL {X  -130.677, Y  +285.194, Z    +0.000, E1   +71.519, E3 +72055.359}
SPL {X  -126.239, Y  +279.212, Z    +0.000, E1   +70.937, E3 +72062.160}
SPL {X  -121.335, Y  +273.218, Z    +0.000, E1   +70.225, E3 +72068.948}
SPL {X   -79.311, Y  +238.552, Z    +0.000, E1   +58.563, E3 +72165.426}
ENDSPLINE

SPLINE
SPL {X  -105.077, Y  +256.854, Z    +0.000, E1   +55.187, E3 +72352.978}
SPL {X  -133.208, Y  +288.886, Z    +0.000, E1   +52.003, E3 +72386.079}
SPL {X  -149.825, Y  +321.381, Z    +0.000, E1   +42.580, E3 +72399.233}
SPL {X  -156.491, Y  +344.222, Z    +0.000, E1   +30.612, E3 +72403.739}
SPL {X  -159.275, Y  +362.387, Z    +0.000, E1   +16.907, E3 +72405.652}
SPL {X  -159.964, Y  +374.630, Z    +0.000, E1    +5.249, E3 +72406.226}
SPL {X  -159.990, Y  +379.484, Z    +0.000, E1    +0.034, E3 +72406.282}
SPL {X  -159.990, Y  +381.639, Z    +0.000, E1    -4.454, E3 +72406.304}
SPL {X  -159.990, Y  +385.871, Z    +0.000, E1   -15.161, E3 +72406.419}
SPL {X  -159.990, Y  +391.065, Z    +0.000, E1   -28.187, E3 +72406.707}
SPL {X  -159.990, Y  +397.286, Z    +0.000, E1   -41.591, E3 +72407.250}
SPL {X  -159.990, Y  +406.369, Z    +0.000, E1   -54.148, E3 +72408.469}
SPL {X  -159.990, Y  +426.617, Z    +0.000, E1   -66.230, E3 +72412.719}
SPL {X  -159.990, Y  +499.521, Z    +0.000, E1   -73.662, E3 +72436.045}
SPL {X  -159.629, Y  +687.249, Z    +0.000, E1   -74.539, E3 +72523.929}
SPL {X  -157.983, Y  +701.765, Z    +0.000, E1   -74.384, E3 +72534.162}
SPL {X  -155.520, Y  +714.054, Z    +0.000, E1   -74.151, E3 +72543.916}
SPL {X  -152.569, Y  +724.660, Z    +0.000, E1   -73.857, E3 +72553.150}
SPL {X  -149.625, Y  +733.149, Z    +0.000, E1   -73.553, E3 +72561.086}
SPL {X  -146.617, Y  +740.532, Z    +0.000, E1   -73.233, E3 +72568.362}
SPL {X  -143.394, Y  +747.457, Z    +0.000, E1   -72.883, E3 +72575.459}
SPL {X  -140.332, Y  +753.336, Z    +0.000, E1   -72.527, E3 +72581.734}
SPL {X  -137.187, Y  +758.820, Z    +0.000, E1   -72.156, E3 +72587.737}
SPL {X  -134.014, Y  +763.891, Z    +0.000, E1   -71.759, E3 +72593.423}
SPL {X  -130.657, Y  +768.834, Z    +0.000, E1   -71.330, E3 +72599.038}
SPL {X  -126.937, Y  +773.885, Z    +0.000, E1   -70.823, E3 +72604.840}
SPL {X  -122.983, Y  +778.833, Z    +0.000, E1   -70.262, E3 +72610.484}
SPL {X  -120.205, Y  +782.082, Z    +0.000, E1   -69.822, E3 +72614.153}
SPL {X   -75.772, Y  +817.409, Z    +0.000, E1   -56.226, E3 +72740.091}
ENDSPLINE

SPLINE
SPL {X  -124.054, Y  +777.532, Z    +0.000, E1   -54.436, E3 +72923.319}
SPL {X  -145.922, Y  +742.101, Z    +0.000, E1   -46.535, E3 +72941.589}
SPL {X  -155.216, Y  +715.293, Z    +0.000, E1   -34.460, E3 +72947.781}
SPL {X  -159.282, Y  +691.530, Z    +0.000, E1   -17.100, E3 +72950.476}
SPL {X  -159.981, Y  +678.202, Z    +0.000, E1    -4.129, E3 +72951.050}
SPL {X  -159.990, Y  +674.500, Z    +0.000, E1    +0.000, E3 +72951.088}
SPL {X  -159.990, Y  +672.677, Z    +0.000, E1    +3.879, E3 +72951.103}
SPL {X  -159.990, Y  +669.117, Z    +0.000, E1   +12.900, E3 +72951.186}
SPL {X  -159.990, Y  +665.253, Z    +0.000, E1   +22.908, E3 +72951.360}
SPL {X  -159.990, Y  +658.335, Z    +0.000, E1   +38.839, E3 +72951.904}
SPL {X  -159.990, Y  +645.786, Z    +0.000, E1   +56.338, E3 +72953.619}
SPL {X  -159.990, Y  +623.264, Z    +0.000, E1   +67.753, E3 +72958.544}
SPL {X  -159.990, Y  +547.268, Z    +0.000, E1   +73.735, E3 +72984.233}
SPL {X  -159.091, Y  +360.560, Z    +0.000, E1   +74.726, E3 +73070.559}
SPL {X  -156.418, Y  +343.879, Z    +0.000, E1   +74.473, E3 +73082.984}
SPL {X  -153.414, Y  +332.103, Z    +0.000, E1   +74.378, E3 +73090.659}
SPL {X  -141.909, Y  +303.617, Z    +0.000, E1   +76.515, E3 +73083.189}
ENDSPLINE

SPLINE
SPL {X  -142.567, Y  +304.895, Z    +0.000, E1   +75.566, E3 +73092.004}
ENDSPLINE

SPLINE
SPL {X  -141.999, Y  +303.790, Z    +0.000, E1   +74.633, E3 +73101.255}
SPL {X  -141.780, Y  +303.371, Z    +0.000, E1   +73.549, E3 +73110.829}
SPL {X  -140.619, Y  +301.190, Z    +0.000, E1   +72.741, E3 +73118.676}
SPL {X  -137.438, Y  +295.601, Z    +0.000, E1   +72.365, E3 +73124.764}
SPL {X  -134.156, Y  +290.328, Z    +0.000, E1   +71.962, E3 +73130.635}
SPL {X  -130.677, Y  +285.194, Z    +0.000, E1   +71.519, E3 +73136.440}
SPL {X  -127.147, Y  +280.390, Z    +0.000, E1   +71.042, E3 +73141.924}
SPL {X  -123.431, Y  +275.709, Z    +0.000, E1   +70.518, E3 +73147.247}
SPL {X  -120.392, Y  +272.131, Z    +0.000, E1   +70.053, E3 +73151.268}
SPL {X   -79.311, Y  +238.552, Z    +0.000, E1   +58.563, E3 +73246.507}
ENDSPLINE

SPLINE
SPL {X  -105.077, Y  +256.854, Z    +0.000, E1   +55.187, E3 +73434.059}
SPL {X  -133.208, Y  +288.886, Z    +0.000, E1   +52.003, E3 +73467.160}
SPL {X  -149.825, Y  +321.381, Z    +0.000, E1   +42.580, E3 +73480.314}
SPL {X  -157.376, Y  +348.695, Z    +0.000, E1   +27.651, E3 +73485.399}
SPL {X  -159.486, Y  +364.808, Z    +0.000, E1   +14.693, E3 +73486.902}
SPL {X  -159.964, Y  +374.630, Z    +0.000, E1    +5.249, E3 +73487.307}
SPL {X  -159.990, Y  +379.484, Z    +0.000, E1    +0.034, E3 +73487.363}
SPL {X  -159.990, Y  +381.639, Z    +0.000, E1    -4.454, E3 +73487.385}
SPL {X  -159.990, Y  +387.459, Z    +0.000, E1   -18.927, E3 +73487.580}
SPL {X  -159.990, Y  +393.138, Z    +0.000, E1   -33.246, E3 +73487.930}
SPL {X  -159.990, Y  +399.326, Z    +0.000, E1   -44.934, E3 +73488.572}
SPL {X  -159.990, Y  +408.817, Z    +0.000, E1   -56.572, E3 +73489.945}
SPL {X  -159.990, Y  +426.617, Z    +0.000, E1   -66.230, E3 +73493.800}
SPL {X  -159.990, Y  +499.521, Z    +0.000, E1   -73.662, E3 +73517.126}
SPL {X  -159.629, Y  +687.249, Z    +0.000, E1   -74.539, E3 +73605.011}
SPL {X  -157.983, Y  +701.765, Z    +0.000, E1   -74.384, E3 +73615.243}
SPL {X  -155.520, Y  +714.054, Z    +0.000, E1   -74.151, E3 +73624.997}
SPL {X  -152.569, Y  +724.660, Z    +0.000, E1   -73.857, E3 +73634.231}
SPL {X  -149.625, Y  +733.149, Z    +0.000, E1   -73.553, E3 +73642.167}
SPL {X  -146.617, Y  +740.532, Z    +0.000, E1   -73.233, E3 +73649.443}
SPL {X  -143.394, Y  +747.457, Z    +0.000, E1   -72.883, E3 +73656.540}
SPL {X  -140.332, Y  +753.336, Z    +0.000, E1   -72.527, E3 +73662.815}
SPL {X  -137.187, Y  +758.820, Z    +0.000, E1   -72.156, E3 +73668.818}
SPL {X  -134.014, Y  +763.891, Z    +0.000, E1   -71.759, E3 +73674.504}
SPL {X  -130.657, Y  +768.834, Z    +0.000, E1   -71.330, E3 +73680.119}
SPL {X  -126.020, Y  +775.068, Z    +0.000, E1   -70.718, E3 +73687.247}
SPL {X  -121.287, Y  +780.838, Z    +0.000, E1   -70.013, E3 +73693.820}
SPL {X   -75.772, Y  +817.409, Z    +0.000, E1   -56.226, E3 +73821.173}
ENDSPLINE

SPLINE
SPL {X  -124.054, Y  +777.532, Z    +0.000, E1   -54.436, E3 +74004.400}
SPL {X  -145.922, Y  +742.101, Z    +0.000, E1   -46.535, E3 +74022.670}
SPL {X  -155.216, Y  +715.293, Z    +0.000, E1   -34.460, E3 +74028.862}
SPL {X  -159.282, Y  +691.530, Z    +0.000, E1   -17.100, E3 +74031.558}
SPL {X  -159.981, Y  +678.202, Z    +0.000, E1    -4.129, E3 +74032.131}
SPL {X  -159.990, Y  +674.500, Z    +0.000, E1    +0.000, E3 +74032.169}
SPL {X  -159.990, Y  +672.677, Z    +0.000, E1    +3.879, E3 +74032.184}
SPL {X  -159.990, Y  +669.117, Z    +0.000, E1   +12.900, E3 +74032.267}
SPL {X  -159.990, Y  +663.639, Z    +0.000, E1   +26.675, E3 +74032.553}
SPL {X  -159.990, Y  +656.057, Z    +0.000, E1   +43.288, E3 +74033.208}
SPL {X  -159.990, Y  +645.786, Z    +0.000, E1   +56.338, E3 +74034.700}
SPL {X  -159.990, Y  +623.264, Z    +0.000, E1   +67.753, E3 +74039.625}
SPL {X  -159.990, Y  +547.268, Z    +0.000, E1   +73.735, E3 +74065.314}
SPL {X  -159.626, Y  +366.721, Z    +0.000, E1   +74.756, E3 +74147.579}
SPL {X  -157.975, Y  +352.185, Z    +0.000, E1   +74.622, E3 +74157.645}
SPL {X  -154.546, Y  +336.120, Z    +0.000, E1   +74.400, E3 +74169.303}
SPL {X  -141.909, Y  +303.617, Z    +0.000, E1   +76.515, E3 +74164.270}
ENDSPLINE

SPLINE
SPL {X  -142.567, Y  +304.895, Z    +0.000, E1   +75.566, E3 +74173.085}
ENDSPLINE

SPLINE
SPL {X  -141.999, Y  +303.790, Z    +0.000, E1   +74.633, E3 +74182.336}
SPL {X  -141.780, Y  +303.371, Z    +0.000, E1   +73.549, E3 +74191.910}
SPL {X  -140.619, Y  +301.190, Z    +0.000, E1   +72.741, E3 +74199.757}
SPL {X  -137.438, Y  +295.601, Z    +0.000, E1   +72.365, E3 +74205.845}
SPL {X  -134.156, Y  +290.328, Z    +0.000, E1   +71.962, E3 +74211.716}
SPL {X  -130.677, Y  +285.194, Z    +0.000, E1   +71.519, E3 +74217.521}
SPL {X  -127.147, Y  +280.390, Z    +0.000, E1   +71.042, E3 +74223.005}
SPL {X  -123.431, Y  +275.709, Z    +0.000, E1   +70.518, E3 +74228.328}
SPL {X  -120.392, Y  +272.131, Z    +0.000, E1   +70.053, E3 +74232.349}
SPL {X   -79.311, Y  +238.552, Z    +0.000, E1   +58.563, E3 +74327.588}
ENDSPLINE

SPLINE
SPL {X  -105.077, Y  +256.854, Z    +0.000, E1   +55.187, E3 +74515.140}
SPL {X  -133.208, Y  +288.886, Z    +0.000, E1   +52.003, E3 +74548.241}
SPL {X  -149.825, Y  +321.381, Z    +0.000, E1   +42.580, E3 +74561.395}
SPL {X  -157.376, Y  +348.695, Z    +0.000, E1   +27.651, E3 +74566.480}
SPL {X  -159.486, Y  +364.808, Z    +0.000, E1   +14.693, E3 +74567.983}
SPL {X  -159.964, Y  +374.630, Z    +0.000, E1    +5.249, E3 +74568.388}
SPL {X  -159.990, Y  +379.484, Z    +0.000, E1    +0.034, E3 +74568.444}
SPL {X  -159.990, Y  +381.639, Z    +0.000, E1    -4.454, E3 +74568.466}
SPL {X  -159.990, Y  +387.459, Z    +0.000, E1   -18.927, E3 +74568.662}
SPL {X  -159.990, Y  +395.361, Z    +0.000, E1   -37.740, E3 +74569.226}
SPL {X  -159.990, Y  +406.369, Z    +0.000, E1   -54.148, E3 +74570.631}
SPL {X  -159.990, Y  +426.617, Z    +0.000, E1   -66.230, E3 +74574.881}
SPL {X  -159.990, Y  +499.521, Z    +0.000, E1   -73.662, E3 +74598.207}
SPL {X  -159.629, Y  +687.249, Z    +0.000, E1   -74.539, E3 +74686.092}
SPL {X  -157.983, Y  +701.765, Z    +0.000, E1   -74.384, E3 +74696.324}
SPL {X  -155.520, Y  +714.054, Z    +0.000, E1   -74.151, E3 +74706.078}
SPL {X  -152.569, Y  +724.660, Z    +0.000, E1   -73.857, E3 +74715.313}
SPL {X  -149.625, Y  +733.149, Z    +0.000, E1   -73.553, E3 +74723.248}
SPL {X  -146.617, Y  +740.532, Z    +0.000, E1   -73.233, E3 +74730.524}
SPL {X  -143.394, Y  +747.457, Z    +0.000, E1   -72.883, E3 +74737.621}
SPL {X  -140.332, Y  +753.336, Z    +0.000, E1   -72.527, E3 +74743.896}
SPL {X  -137.187, Y  +758.820, Z    +0.000, E1   -72.156, E3 +74749.899}
SPL {X  -134.014, Y  +763.891, Z    +0.000, E1   -71.759, E3 +74755.585}
SPL {X  -130.657, Y  +768.834, Z    +0.000, E1   -71.330, E3 +74761.200}
SPL {X  -126.937, Y  +773.885, Z    +0.000, E1   -70.823, E3 +74767.002}
SPL {X  -122.983, Y  +778.833, Z    +0.000, E1   -70.262, E3 +74772.646}
SPL {X  -120.205, Y  +782.082, Z    +0.000, E1   -69.822, E3 +74776.315}
SPL {X   -77.717, Y  +816.346, Z    +0.000, E1   -57.422, E3 +74884.166}
SPL {X   -74.440, Y  +818.117, Z    +0.000, E1   -54.647, E3 +74937.405}
ENDSPLINE

SPLINE
SPL {X  -124.054, Y  +777.532, Z    +0.000, E1   -54.436, E3 +75085.481}
SPL {X  -149.719, Y  +732.901, Z    +0.000, E1   -43.150, E3 +75106.296}
SPL {X  -158.004, Y  +701.630, Z    +0.000, E1   -25.366, E3 +75111.760}
SPL {X  -159.838, Y  +683.473, Z    +0.000, E1    -9.532, E3 +75113.067}
SPL {X  -159.990, Y  +674.579, Z    +0.000, E1    -0.168, E3 +75113.250}
SPL {X  -159.990, Y  +672.677, Z    +0.000, E1    +3.879, E3 +75113.265}
SPL {X  -159.990, Y  +669.117, Z    +0.000, E1   +12.900, E3 +75113.348}
SPL {X  -159.990, Y  +665.253, Z    +0.000, E1   +22.908, E3 +75113.522}
SPL {X  -159.990, Y  +658.335, Z    +0.000, E1   +38.839, E3 +75114.066}
SPL {X  -159.990, Y  +645.786, Z    +0.000, E1   +56.338, E3 +75115.781}
SPL {X  -159.990, Y  +623.264, Z    +0.000, E1   +67.753, E3 +75120.707}
SPL {X  -159.990, Y  +547.268, Z    +0.000, E1   +73.735, E3 +75146.395}
SPL {X  -159.091, Y  +360.560, Z    +0.000, E1   +74.726, E3 +75232.721}
SPL {X  -156.418, Y  +343.879, Z    +0.000, E1   +74.473, E3 +75245.146}
SPL {X  -153.414, Y  +332.103, Z    +0.000, E1   +74.378, E3 +75252.821}
SPL {X  -141.909, Y  +303.617, Z    +0.000, E1   +76.515, E3 +75245.351}
ENDSPLINE

SPLINE
SPL {X  -142.567, Y  +304.895, Z    +0.000, E1   +75.566, E3 +75254.166}
ENDSPLINE

SPLINE
SPL {X  -141.999, Y  +303.790, Z    +0.000, E1   +74.633, E3 +75263.418}
SPL {X  -141.780, Y  +303.371, Z    +0.000, E1   +73.549, E3 +75272.991}
SPL {X  -140.619, Y  +301.190, Z    +0.000, E1   +72.741, E3 +75280.838}
SPL {X  -137.438, Y  +295.601, Z    +0.000, E1   +72.365, E3 +75286.926}
SPL {X  -134.156, Y  +290.328, Z    +0.000, E1   +71.962, E3 +75292.797}
SPL {X  -130.677, Y  +285.194, Z    +0.000, E1   +71.519, E3 +75298.602}
SPL {X  -127.147, Y  +280.390, Z    +0.000, E1   +71.042, E3 +75304.086}
SPL {X  -123.431, Y  +275.709, Z    +0.000, E1   +70.518, E3 +75309.409}
SPL {X  -120.392, Y  +272.131, Z    +0.000, E1   +70.053, E3 +75313.430}
SPL {X   -79.311, Y  +238.552, Z    +0.000, E1   +58.563, E3 +75408.669}
ENDSPLINE

SPLINE
SPL {X  -105.077, Y  +256.854, Z    +0.000, E1   +55.187, E3 +75596.221}
SPL {X  -133.208, Y  +288.886, Z    +0.000, E1   +52.003, E3 +75629.322}
SPL {X  -149.825, Y  +321.381, Z    +0.000, E1   +42.580, E3 +75642.476}
SPL {X  -157.376, Y  +348.695, Z    +0.000, E1   +27.651, E3 +75647.561}
SPL {X  -159.486, Y  +364.808, Z    +0.000, E1   +14.693, E3 +75649.064}
SPL {X  -159.964, Y  +374.630, Z    +0.000, E1    +5.249, E3 +75649.469}
SPL {X  -159.990, Y  +379.735, Z    +0.000, E1    -0.236, E3 +75649.526}
SPL {X  -159.990, Y  +384.648, Z    +0.000, E1   -11.739, E3 +75649.623}
SPL {X  -159.990, Y  +391.065, Z    +0.000, E1   -28.187, E3 +75649.951}
SPL {X  -159.990, Y  +399.326, Z    +0.000, E1   -44.934, E3 +75650.734}
SPL {X  -159.990, Y  +408.817, Z    +0.000, E1   -56.572, E3 +75652.107}
SPL {X  -159.990, Y  +426.617, Z    +0.000, E1   -66.230, E3 +75655.962}
SPL {X  -159.990, Y  +499.521, Z    +0.000, E1   -73.662, E3 +75679.289}
SPL {X  -159.629, Y  +687.249, Z    +0.000, E1   -74.539, E3 +75767.173}
SPL {X  -157.983, Y  +701.765, Z    +0.000, E1   -74.384, E3 +75777.405}
SPL {X  -155.520, Y  +714.054, Z    +0.000, E1   -74.151, E3 +75787.159}
SPL {X  -152.569, Y  +724.660, Z    +0.000, E1   -73.857, E3 +75796.394}
SPL {X  -149.625, Y  +733.149, Z    +0.000, E1   -73.553, E3 +75804.329}
SPL {X  -146.617, Y  +740.532, Z    +0.000, E1   -73.233, E3 +75811.605}
SPL {X  -143.394, Y  +747.457, Z    +0.000, E1   -72.883, E3 +75818.702}
SPL {X  -140.332, Y  +753.336, Z    +0.000, E1   -72.527, E3 +75824.977}
SPL {X  -137.187, Y  +758.820, Z    +0.000, E1   -72.156, E3 +75830.980}
SPL {X  -134.014, Y  +763.891, Z    +0.000, E1   -71.759, E3 +75836.666}
SPL {X  -130.657, Y  +768.834, Z    +0.000, E1   -71.330, E3 +75842.281}
SPL {X  -126.020, Y  +775.068, Z    +0.000, E1   -70.718, E3 +75849.409}
SPL {X  -121.287, Y  +780.838, Z    +0.000, E1   -70.013, E3 +75855.982}
SPL {X   -75.772, Y  +817.409, Z    +0.000, E1   -56.226, E3 +75983.335}
ENDSPLINE

SPLINE
SPL {X  -124.054, Y  +777.532, Z    +0.000, E1   -54.436, E3 +76166.563}
SPL {X  -149.719, Y  +732.901, Z    +0.000, E1   -43.150, E3 +76187.377}
SPL {X  -158.004, Y  +701.630, Z    +0.000, E1   -25.366, E3 +76192.842}
SPL {X  -159.639, Y  +687.095, Z    +0.000, E1   -12.931, E3 +76194.000}
SPL {X  -159.981, Y  +678.202, Z    +0.000, E1    -4.129, E3 +76194.294}
SPL {X  -159.990, Y  +674.500, Z    +0.000, E1    +0.000, E3 +76194.331}
SPL {X  -159.990, Y  +672.677, Z    +0.000, E1    +3.879, E3 +76194.347}
SPL {X  -159.990, Y  +669.117, Z    +0.000, E1   +12.900, E3 +76194.429}
SPL {X  -159.990, Y  +663.639, Z    +0.000, E1   +26.675, E3 +76194.715}
SPL {X  -159.990, Y  +656.057, Z    +0.000, E1   +43.288, E3 +76195.371}
SPL {X  -159.990, Y  +645.786, Z    +0.000, E1   +56.338, E3 +76196.862}
SPL {X  -159.990, Y  +623.264, Z    +0.000, E1   +67.753, E3 +76201.788}
SPL {X  -159.990, Y  +547.268, Z    +0.000, E1   +73.735, E3 +76227.476}
SPL {X  -159.091, Y  +360.560, Z    +0.000, E1   +74.726, E3 +76313.802}
SPL {X  -156.418, Y  +343.879, Z    +0.000, E1   +74.473, E3 +76326.228}
SPL {X  -153.414, Y  +332.103, Z    +0.000, E1   +74.378, E3 +76333.902}
SPL {X  -141.909, Y  +303.617, Z    +0.000, E1   +76.515, E3 +76326.432}
ENDSPLINE

SPLINE
SPL {X  -142.567, Y  +304.895, Z    +0.000, E1   +75.566, E3 +76335.247}
ENDSPLINE

SPLINE
SPL {X  -141.999, Y  +303.790, Z    +0.000, E1   +74.633, E3 +76344.499}
SPL {X  -141.780, Y  +303.371, Z    +0.000, E1   +73.549, E3 +76354.072}
SPL {X  -140.619, Y  +301.190, Z    +0.000, E1   +72.741, E3 +76361.919}
SPL {X  -137.438, Y  +295.601, Z    +0.000, E1   +72.365, E3 +76368.007}
SPL {X  -134.156, Y  +290.328, Z    +0.000, E1   +71.962, E3 +76373.878}
SPL {X  -130.677, Y  +285.194, Z    +0.000, E1   +71.519, E3 +76379.683}
SPL {X  -127.147, Y  +280.390, Z    +0.000, E1   +71.042, E3 +76385.167}
SPL {X  -123.431, Y  +275.709, Z    +0.000, E1   +70.518, E3 +76390.490}
SPL {X  -120.392, Y  +272.131, Z    +0.000, E1   +70.053, E3 +76394.511}
SPL {X   -79.311, Y  +238.552, Z    +0.000, E1   +58.563, E3 +76489.750}
ENDSPLINE

SPLINE
SPL {X  -105.077, Y  +256.854, Z    +0.000, E1   +55.187, E3 +76677.302}
SPL {X  -133.208, Y  +288.886, Z    +0.000, E1   +52.003, E3 +76710.403}
SPL {X  -149.825, Y  +321.381, Z    +0.000, E1   +42.580, E3 +76723.557}
SPL {X  -157.376, Y  +348.695, Z    +0.000, E1   +27.651, E3 +76728.642}
SPL {X  -159.486, Y  +364.808, Z    +0.000, E1   +14.693, E3 +76730.145}
SPL {X  -159.964, Y  +374.630, Z    +0.000, E1    +5.249, E3 +76730.550}
SPL {X  -159.990, Y  +379.484, Z    +0.000, E1    +0.034, E3 +76730.606}
SPL {X  -159.990, Y  +381.639, Z    +0.000, E1    -4.454, E3 +76730.628}
SPL {X  -159.990, Y  +387.459, Z    +0.000, E1   -18.927, E3 +76730.824}
SPL {X  -159.990, Y  +393.138, Z    +0.000, E1   -33.246, E3 +76731.173}
SPL {X  -159.990, Y  +399.326, Z    +0.000, E1   -44.934, E3 +76731.815}
SPL {X  -159.990, Y  +408.817, Z    +0.000, E1   -56.572, E3 +76733.188}
SPL {X  -159.990, Y  +426.617, Z    +0.000, E1   -66.230, E3 +76737.043}
SPL {X  -159.990, Y  +499.521, Z    +0.000, E1   -73.662, E3 +76760.370}
SPL {X  -159.629, Y  +687.249, Z    +0.000, E1   -74.539, E3 +76848.254}
SPL {X  -157.983, Y  +701.765, Z    +0.000, E1   -74.384, E3 +76858.486}
SPL {X  -155.520, Y  +714.054, Z    +0.000, E1   -74.151, E3 +76868.240}
SPL {X  -152.569, Y  +724.660, Z    +0.000, E1   -73.857, E3 +76877.475}
SPL {X  -149.625, Y  +733.149, Z    +0.000, E1   -73.553, E3 +76885.410}
SPL {X  -146.617, Y  +740.532, Z    +0.000, E1   -73.233, E3 +76892.686}
SPL {X  -143.394, Y  +747.457, Z    +0.000, E1   -72.883, E3 +76899.783}
SPL {X  -140.332, Y  +753.336, Z    +0.000, E1   -72.527, E3 +76906.058}
SPL {X  -137.187, Y  +758.820, Z    +0.000, E1   -72.156, E3 +76912.061}
SPL {X  -134.014, Y  +763.891, Z    +0.000, E1   -71.759, E3 +76917.747}
SPL {X  -130.657, Y  +768.834, Z    +0.000, E1   -71.330, E3 +76923.362}
SPL {X  -126.937, Y  +773.885, Z    +0.000, E1   -70.823, E3 +76929.164}
SPL {X  -122.983, Y  +778.833, Z    +0.000, E1   -70.262, E3 +76934.809}
SPL {X  -120.205, Y  +782.082, Z    +0.000, E1   -69.822, E3 +76938.477}
SPL {X   -75.772, Y  +817.409, Z    +0.000, E1   -56.226, E3 +77064.416}
ENDSPLINE

SPLINE
SPL {X  -124.054, Y  +777.532, Z    +0.000, E1   -54.436, E3 +77247.644}
SPL {X  -145.922, Y  +742.101, Z    +0.000, E1   -46.535, E3 +77265.913}
SPL {X  -155.216, Y  +715.293, Z    +0.000, E1   -34.460, E3 +77272.106}
SPL {X  -159.282, Y  +691.530, Z    +0.000, E1   -17.100, E3 +77274.801}
SPL {X  -159.981, Y  +678.202, Z    +0.000, E1    -4.129, E3 +77275.375}
SPL {X  -159.990, Y  +674.500, Z    +0.000, E1    +0.000, E3 +77275.412}
SPL {X  -159.990, Y  +672.677, Z    +0.000, E1    +3.879, E3 +77275.428}
SPL {X  -159.990, Y  +669.117, Z    +0.000, E1   +12.900, E3 +77275.510}
SPL {X  -159.990, Y  +665.253, Z    +0.000, E1   +22.908, E3 +77275.684}
SPL {X  -159.990, Y  +658.335, Z    +0.000, E1   +38.839, E3 +77276.229}
SPL {X  -159.990, Y  +645.786, Z    +0.000, E1   +56.338, E3 +77277.943}
SPL {X  -159.990, Y  +623.264, Z    +0.000, E1   +67.753, E3 +77282.869}
SPL {X  -159.990, Y  +547.268, Z    +0.000, E1   +73.735, E3 +77308.557}
SPL {X  -159.091, Y  +360.560, Z    +0.000, E1   +74.726, E3 +77394.883}
SPL {X  -156.418, Y  +343.879, Z    +0.000, E1   +74.473, E3 +77407.309}
SPL {X  -153.414, Y  +332.103, Z    +0.000, E1   +74.378, E3 +77414.983}
SPL {X  -141.909, Y  +303.617, Z    +0.000, E1   +76.515, E3 +77407.513}
ENDSPLINE

SPLINE
SPL {X  -142.567, Y  +304.895, Z    +0.000, E1   +75.566, E3 +77416.328}
ENDSPLINE

SPLINE
SPL {X  -141.999, Y  +303.790, Z    +0.000, E1   +74.633, E3 +77425.580}
SPL {X  -141.780, Y  +303.371, Z    +0.000, E1   +73.549, E3 +77435.153}
SPL {X  -140.619, Y  +301.190, Z    +0.000, E1   +72.741, E3 +77443.000}
SPL {X  -137.438, Y  +295.601, Z    +0.000, E1   +72.365, E3 +77449.088}
SPL {X  -134.156, Y  +290.328, Z    +0.000, E1   +71.962, E3 +77454.959}
SPL {X  -130.677, Y  +285.194, Z    +0.000, E1   +71.519, E3 +77460.764}
SPL {X  -126.239, Y  +279.212, Z    +0.000, E1   +70.937, E3 +77467.565}
SPL {X  -121.335, Y  +273.218, Z    +0.000, E1   +70.225, E3 +77474.354}
SPL {X   -79.311, Y  +238.552, Z    +0.000, E1   +58.563, E3 +77570.831}
ENDSPLINE

SPLINE
SPL {X  -105.077, Y  +256.854, Z    +0.000, E1   +55.187, E3 +77758.383}
SPL {X  -133.208, Y  +288.886, Z    +0.000, E1   +52.003, E3 +77791.484}
SPL {X  -149.825, Y  +321.381, Z    +0.000, E1   +42.580, E3 +77804.638}
SPL {X  -157.376, Y  +348.695, Z    +0.000, E1   +27.651, E3 +77809.723}
SPL {X  -159.486, Y  +364.808, Z    +0.000, E1   +14.693, E3 +77811.226}
SPL {X  -159.964, Y  +374.630, Z    +0.000, E1    +5.249, E3 +77811.631}
SPL {X  -159.990, Y  +379.484, Z    +0.000, E1    +0.034, E3 +77811.687}
SPL {X  -159.990, Y  +381.639, Z    +0.000, E1    -4.454, E3 +77811.709}
SPL {X  -159.990, Y  +385.871, Z    +0.000, E1   -15.161, E3 +77811.825}
SPL {X  -159.990, Y  +391.065, Z    +0.000, E1   -28.187, E3 +77812.113}
SPL {X  -159.990, Y  +399.326, Z    +0.000, E1   -44.934, E3 +77812.896}
SPL {X  -159.990, Y  +408.817, Z    +0.000, E1   -56.572, E3 +77814.269}
SPL {X  -159.990, Y  +426.617, Z    +0.000, E1   -66.230, E3 +77818.124}
SPL {X  -159.990, Y  +499.521, Z    +0.000, E1   -73.662, E3 +77841.451}
SPL {X  -159.629, Y  +687.249, Z    +0.000, E1   -74.539, E3 +77929.335}
SPL {X  -157.983, Y  +701.765, Z    +0.000, E1   -74.384, E3 +77939.567}
SPL {X  -155.520, Y  +714.054, Z    +0.000, E1   -74.151, E3 +77949.321}
SPL {X  -152.569, Y  +724.660, Z    +0.000, E1   -73.857, E3 +77958.556}
SPL {X  -149.625, Y  +733.149, Z    +0.000, E1   -73.553, E3 +77966.491}
SPL {X  -146.617, Y  +740.532, Z    +0.000, E1   -73.233, E3 +77973.767}
SPL {X  -143.394, Y  +747.457, Z    +0.000, E1   -72.883, E3 +77980.864}
SPL {X  -140.332, Y  +753.336, Z    +0.000, E1   -72.527, E3 +77987.139}
SPL {X  -137.187, Y  +758.820, Z    +0.000, E1   -72.156, E3 +77993.142}
SPL {X  -134.014, Y  +763.891, Z    +0.000, E1   -71.759, E3 +77998.828}
SPL {X  -130.657, Y  +768.834, Z    +0.000, E1   -71.330, E3 +78004.443}
SPL {X  -126.020, Y  +775.068, Z    +0.000, E1   -70.718, E3 +78011.571}
SPL {X  -121.287, Y  +780.838, Z    +0.000, E1   -70.013, E3 +78018.145}
SPL {X   -75.772, Y  +817.409, Z    +0.000, E1   -56.226, E3 +78145.497}
ENDSPLINE

SPLINE
SPL {X  -124.054, Y  +777.532, Z    +0.000, E1   -54.436, E3 +78328.725}
SPL {X  -145.922, Y  +742.101, Z    +0.000, E1   -46.535, E3 +78346.994}
SPL {X  -155.216, Y  +715.293, Z    +0.000, E1   -34.460, E3 +78353.187}
SPL {X  -159.282, Y  +691.530, Z    +0.000, E1   -17.100, E3 +78355.882}
SPL {X  -159.981, Y  +678.202, Z    +0.000, E1    -4.129, E3 +78356.456}
SPL {X  -159.990, Y  +674.500, Z    +0.000, E1    +0.000, E3 +78356.493}
SPL {X  -159.990, Y  +672.677, Z    +0.000, E1    +3.879, E3 +78356.509}
SPL {X  -159.990, Y  +669.117, Z    +0.000, E1   +12.900, E3 +78356.591}
SPL {X  -159.990, Y  +663.639, Z    +0.000, E1   +26.675, E3 +78356.877}
SPL {X  -159.990, Y  +656.057, Z    +0.000, E1   +43.288, E3 +78357.533}
SPL {X  -159.990, Y  +647.797, Z    +0.000, E1   +54.469, E3 +78358.670}
SPL {X  -159.990, Y  +630.178, Z    +0.000, E1   +65.480, E3 +78362.354}
SPL {X  -159.990, Y  +547.268, Z    +0.000, E1   +73.735, E3 +78389.638}
SPL {X  -159.626, Y  +366.721, Z    +0.000, E1   +74.756, E3 +78471.903}
SPL {X  -158.582, Y  +356.317, Z    +0.000, E1   +74.662, E3 +78478.996}
SPL {X  -156.418, Y  +343.879, Z    +0.000, E1   +74.473, E3 +78488.390}
SPL {X  -153.414, Y  +332.103, Z    +0.000, E1   +74.378, E3 +78496.064}
SPL {X  -141.909, Y  +303.617, Z    +0.000, E1   +76.515, E3 +78488.594}
ENDSPLINE

SPLINE
SPL {X  -142.567, Y  +304.895, Z    +0.000, E1   +75.566, E3 +78497.410}
ENDSPLINE

SPLINE
SPL {X  -141.999, Y  +303.790, Z    +0.000, E1   +74.633, E3 +78506.661}
SPL {X  -141.780, Y  +303.371, Z    +0.000, E1   +73.549, E3 +78516.235}
SPL {X  -140.619, Y  +301.190, Z    +0.000, E1   +72.741, E3 +78524.081}
SPL {X  -137.438, Y  +295.601, Z    +0.000, E1   +72.365, E3 +78530.169}
SPL {X  -134.156, Y  +290.328, Z    +0.000, E1   +71.962, E3 +78536.040}
SPL {X  -130.677, Y  +285.194, Z    +0.000, E1   +71.519, E3 +78541.846}
SPL {X  -126.239, Y  +279.212, Z    +0.000, E1   +70.937, E3 +78548.647}
SPL {X  -121.335, Y  +273.218, Z    +0.000, E1   +70.225, E3 +78555.435}
SPL {X   -79.311, Y  +238.552, Z    +0.000, E1   +58.563, E3 +78651.912}
ENDSPLINE

SPLINE
SPL {X  -105.077, Y  +256.854, Z    +0.000, E1   +55.187, E3 +78839.464}
SPL {X  -133.208, Y  +288.886, Z    +0.000, E1   +52.003, E3 +78872.565}
SPL {X  -149.825, Y  +321.381, Z    +0.000, E1   +42.580, E3 +78885.719}
SPL {X  -156.491, Y  +344.222, Z    +0.000, E1   +30.612, E3 +78890.225}
SPL {X  -159.275, Y  +362.387, Z    +0.000, E1   +16.907, E3 +78892.139}
SPL {X  -159.964, Y  +374.630, Z    +0.000, E1    +5.249, E3 +78892.712}
SPL {X  -159.990, Y  +379.484, Z    +0.000, E1    +0.034, E3 +78892.768}
SPL {X  -159.990, Y  +381.639, Z    +0.000, E1    -4.454, E3 +78892.790}
SPL {X  -159.990, Y  +385.871, Z    +0.000, E1   -15.161, E3 +78892.906}
SPL {X  -159.990, Y  +391.065, Z    +0.000, E1   -28.187, E3 +78893.194}
SPL {X  -159.990, Y  +399.326, Z    +0.000, E1   -44.934, E3 +78893.977}
SPL {X  -159.990, Y  +408.817, Z    +0.000, E1   -56.572, E3 +78895.350}
SPL {X  -159.990, Y  +426.617, Z    +0.000, E1   -66.230, E3 +78899.205}
SPL {X  -159.990, Y  +499.521, Z    +0.000, E1   -73.662, E3 +78922.532}
SPL {X  -159.629, Y  +687.249, Z    +0.000, E1   -74.539, E3 +79010.416}
SPL {X  -157.983, Y  +701.765, Z    +0.000, E1   -74.384, E3 +79020.648}
SPL {X  -155.520, Y  +714.054, Z    +0.000, E1   -74.151, E3 +79030.402}
SPL {X  -152.569, Y  +724.660, Z    +0.000, E1   -73.857, E3 +79039.637}
SPL {X  -149.625, Y  +733.149, Z    +0.000, E1   -73.553, E3 +79047.572}
SPL {X  -146.617, Y  +740.532, Z    +0.000, E1   -73.233, E3 +79054.848}
SPL {X  -143.394, Y  +747.457, Z    +0.000, E1   -72.883, E3 +79061.945}
SPL {X  -140.332, Y  +753.336, Z    +0.000, E1   -72.527, E3 +79068.220}
SPL {X  -137.187, Y  +758.820, Z    +0.000, E1   -72.156, E3 +79074.223}
SPL {X  -134.014, Y  +763.891, Z    +0.000, E1   -71.759, E3 +79079.909}
SPL {X  -130.657, Y  +768.834, Z    +0.000, E1   -71.330, E3 +79085.524}
SPL {X  -126.937, Y  +773.885, Z    +0.000, E1   -70.823, E3 +79091.326}
SPL {X  -122.983, Y  +778.833, Z    +0.000, E1   -70.262, E3 +79096.971}
SPL {X  -120.205, Y  +782.082, Z    +0.000, E1   -69.822, E3 +79100.639}
SPL {X   -75.772, Y  +817.409, Z    +0.000, E1   -56.226, E3 +79226.578}
ENDSPLINE

SPLINE
SPL {X  -124.054, Y  +777.532, Z    +0.000, E1   -54.436, E3 +79409.806}
SPL {X  -145.922, Y  +742.101, Z    +0.000, E1   -46.535, E3 +79428.075}
SPL {X  -155.216, Y  +715.293, Z    +0.000, E1   -34.460, E3 +79434.268}
SPL {X  -159.282, Y  +691.530, Z    +0.000, E1   -17.100, E3 +79436.963}
SPL {X  -159.981, Y  +678.202, Z    +0.000, E1    -4.129, E3 +79437.537}
SPL {X  -159.990, Y  +674.500, Z    +0.000, E1    +0.000, E3 +79437.574}
SPL {X  -159.990, Y  +672.677, Z    +0.000, E1    +3.879, E3 +79437.590}
SPL {X  -159.990, Y  +669.117, Z    +0.000, E1   +12.900, E3 +79437.672}
SPL {X  -159.990, Y  +665.253, Z    +0.000, E1   +22.908, E3 +79437.846}
SPL {X  -159.990, Y  +658.335, Z    +0.000, E1   +38.839, E3 +79438.391}
SPL {X  -159.990, Y  +645.786, Z    +0.000, E1   +56.338, E3 +79440.105}
SPL {X  -159.990, Y  +623.264, Z    +0.000, E1   +67.753, E3 +79445.031}
SPL {X  -159.990, Y  +547.268, Z    +0.000, E1   +73.735, E3 +79470.719}
SPL {X  -159.091, Y  +360.560, Z    +0.000, E1   +74.726, E3 +79557.045}
SPL {X  -156.418, Y  +343.879, Z    +0.000, E1   +74.473, E3 +79569.471}
SPL {X  -153.414, Y  +332.103, Z    +0.000, E1   +74.378, E3 +79577.146}
SPL {X  -141.909, Y  +303.617, Z    +0.000, E1   +76.515, E3 +79569.676}
ENDSPLINE

SPLINE
SPL {X  -142.567, Y  +304.895, Z    +0.000, E1   +75.566, E3 +79578.491}
ENDSPLINE

SPLINE
SPL {X  -141.999, Y  +303.790, Z    +0.000, E1   +74.633, E3 +79587.742}
SPL {X  -141.780, Y  +303.371, Z    +0.000, E1   +73.549, E3 +79597.316}
SPL {X  -140.619, Y  +301.190, Z    +0.000, E1   +72.741, E3 +79605.162}
SPL {X  -137.438, Y  +295.601, Z    +0.000, E1   +72.365, E3 +79611.251}
SPL {X  -134.156, Y  +290.328, Z    +0.000, E1   +71.962, E3 +79617.122}
SPL {X  -130.677, Y  +285.194, Z    +0.000, E1   +71.519, E3 +79622.927}
SPL {X  -127.147, Y  +280.390, Z    +0.000, E1   +71.042, E3 +79628.411}
SPL {X  -123.431, Y  +275.709, Z    +0.000, E1   +70.518, E3 +79633.734}
SPL {X  -120.392, Y  +272.131, Z    +0.000, E1   +70.053, E3 +79637.754}
SPL {X   -79.311, Y  +238.552, Z    +0.000, E1   +58.563, E3 +79732.993}
ENDSPLINE

SPLINE
SPL {X  -105.077, Y  +256.854, Z    +0.000, E1   +55.187, E3 +79920.545}
SPL {X  -133.208, Y  +288.886, Z    +0.000, E1   +52.003, E3 +79953.647}
SPL {X  -149.825, Y  +321.381, Z    +0.000, E1   +42.580, E3 +79966.800}
SPL {X  -157.376, Y  +348.695, Z    +0.000, E1   +27.651, E3 +79971.885}
SPL {X  -159.486, Y  +364.808, Z    +0.000, E1   +14.693, E3 +79973.388}
SPL {X  -159.964, Y  +374.630, Z    +0.000, E1    +5.249, E3 +79973.793}
SPL {X  -159.990, Y  +379.484, Z    +0.000, E1    +0.034, E3 +79973.849}
SPL {X  -159.990, Y  +381.639, Z    +0.000, E1    -4.454, E3 +79973.871}
SPL {X  -159.990, Y  +387.459, Z    +0.000, E1   -18.927, E3 +79974.067}
SPL {X  -159.990, Y  +393.138, Z    +0.000, E1   -33.246, E3 +79974.416}
SPL {X  -159.990, Y  +399.326, Z    +0.000, E1   -44.934, E3 +79975.058}
SPL {X  -159.990, Y  +408.817, Z    +0.000, E1   -56.572, E3 +79976.431}
SPL {X  -159.990, Y  +426.617, Z    +0.000, E1   -66.230, E3 +79980.286}
SPL {X  -159.990, Y  +499.521, Z    +0.000, E1   -73.662, E3 +80003.613}
SPL {X  -159.629, Y  +687.249, Z    +0.000, E1   -74.539, E3 +80091.497}
SPL {X  -157.983, Y  +701.765, Z    +0.000, E1   -74.384, E3 +80101.729}
SPL {X  -155.520, Y  +714.054, Z    +0.000, E1   -74.151, E3 +80111.483}
SPL {X  -152.569, Y  +724.660, Z    +0.000, E1   -73.857, E3 +80120.718}
SPL {X  -149.625, Y  +733.149, Z    +0.000, E1   -73.553, E3 +80128.653}
SPL {X  -146.617, Y  +740.532, Z    +0.000, E1   -73.233, E3 +80135.930}
SPL {X  -143.394, Y  +747.457, Z    +0.000, E1   -72.883, E3 +80143.027}
SPL {X  -140.332, Y  +753.336, Z    +0.000, E1   -72.527, E3 +80149.301}
SPL {X  -137.187, Y  +758.820, Z    +0.000, E1   -72.156, E3 +80155.305}
SPL {X  -134.014, Y  +763.891, Z    +0.000, E1   -71.759, E3 +80160.990}
SPL {X  -130.657, Y  +768.834, Z    +0.000, E1   -71.330, E3 +80166.605}
SPL {X  -126.937, Y  +773.885, Z    +0.000, E1   -70.823, E3 +80172.407}
SPL {X  -122.983, Y  +778.833, Z    +0.000, E1   -70.262, E3 +80178.052}
SPL {X  -120.205, Y  +782.082, Z    +0.000, E1   -69.822, E3 +80181.720}
SPL {X   -75.772, Y  +817.409, Z    +0.000, E1   -56.226, E3 +80307.659}
ENDSPLINE

